C01810=1020.212,130.588,385.207,167.534,51.338,159.515
C01811=1020.208,130.339,385.227,167.532,51.345,159.516
C01812=1020.202,130.090,385.246,167.528,51.352,159.517
C01813=1020.197,129.841,385.267,167.525,51.359,159.518
C01814=1020.191,129.591,385.286,167.522,51.366,159.518
C01815=1020.186,129.343,385.305,167.520,51.373,159.519
C01816=1020.180,129.093,385.324,167.516,51.380,159.520
C01817=1020.175,128.844,385.343,167.513,51.387,159.521
C01818=1020.169,128.595,385.362,167.510,51.394,159.522
C01819=1020.164,128.346,385.381,167.506,51.401,159.522
C01820=1020.158,128.096,385.401,167.504,51.407,159.523
C01821=1020.153,127.847,385.419,167.501,51.415,159.524
C01822=1020.148,127.598,385.439,167.498,51.422,159.525
C01823=1020.142,127.348,385.459,167.495,51.429,159.526
C01824=1020.137,127.099,385.477,167.491,51.436,159.527
C01825=1020.132,126.850,385.497,167.489,51.442,159.528
C01826=1020.126,126.601,385.516,167.486,51.450,159.529
C01827=1020.121,126.352,385.535,167.483,51.457,159.529
C01828=1020.115,126.102,385.554,167.479,51.464,159.530
C01829=1020.109,125.853,385.573,167.477,51.470,159.531
C01830=1020.104,125.604,385.592,167.474,51.477,159.532
C01831=1020.099,125.355,385.611,167.470,51.484,159.533
C01832=1020.094,125.106,385.630,167.467,51.491,159.533
C01833=1020.089,124.856,385.650,167.465,51.498,159.534
C01834=1020.083,124.607,385.669,167.462,51.505,159.535
C01835=1020.078,124.358,385.688,167.459,51.512,159.536
C01836=1020.072,124.109,385.707,167.455,51.519,159.537
C01837=1020.067,123.860,385.726,167.453,51.526,159.538
C01838=1020.061,123.577,385.748,167.449,51.534,159.538
C01839=1020.054,123.294,385.770,167.446,51.541,159.539
C01840=1020.048,123.011,385.792,167.442,51.549,159.540
C01841=1020.042,122.729,385.813,167.439,51.557,159.541
C01842=1020.037,122.480,385.832,167.436,51.564,159.542
C01843=1020.032,122.230,385.852,167.433,51.571,159.543
C01844=1020.027,121.982,385.871,167.430,51.578,159.544
C01845=1020.021,121.732,385.890,167.428,51.585,159.545
C01846=1020.016,121.484,385.909,167.424,51.592,159.545
C01847=1020.010,121.234,385.928,167.421,51.599,159.546
C01848=1020.005,120.985,385.946,167.419,51.606,159.547
C01849=1020.000,120.735,385.965,167.416,51.612,159.548
C01850=1019.994,120.486,385.985,167.412,51.619,159.549
C01851=1019.989,120.237,386.003,167.410,51.626,159.550
C01852=1019.983,119.988,386.023,167.407,51.633,159.550
C01853=1019.978,119.739,386.042,167.403,51.640,159.551
C01854=1019.972,119.490,386.061,167.401,51.647,159.552
C01855=1019.968,119.240,386.080,167.398,51.654,159.553
C01856=1019.963,118.990,386.099,167.395,51.660,159.554
C01857=1019.958,118.742,386.118,167.392,51.667,159.554
C01858=1019.952,118.492,386.137,167.389,51.675,159.555
C01859=1019.947,118.244,386.156,167.386,51.682,159.556
C01860=1019.941,117.993,386.174,167.384,51.688,159.557
C01861=1019.936,117.745,386.193,167.381,51.695,159.558
C01862=1019.931,117.495,386.212,167.377,51.702,159.559
C01863=1019.926,117.247,386.231,167.375,51.709,159.560
C01864=1019.920,116.997,386.251,167.372,51.716,159.560
C01865=1019.915,116.748,386.269,167.369,51.723,159.561
C01866=1019.909,116.498,386.288,167.366,51.729,159.562
C01867=1019.904,116.250,386.307,167.363,51.736,159.563
C01868=1019.899,116.001,386.326,167.361,51.743,159.564
C01869=1019.894,115.751,386.344,167.358,51.750,159.564
C01870=1019.890,115.502,386.364,167.354,51.757,159.565
C01871=1019.884,115.252,386.383,167.352,51.764,159.566
C01872=1019.879,115.004,386.402,167.349,51.771,159.567
C01873=1019.873,114.754,386.420,167.345,51.778,159.568
C01874=1019.868,114.505,386.439,167.343,51.784,159.568
C01875=1019.863,114.255,386.459,167.340,51.791,159.569
C01876=1019.858,114.006,386.477,167.338,51.798,159.570
C01877=1019.853,113.757,386.496,167.334,51.804,159.571
C01878=1019.847,113.508,386.515,167.332,51.811,159.572
C01879=1019.842,113.259,386.533,167.329,51.818,159.572
C01880=1019.837,113.009,386.552,167.325,51.825,159.573
C01881=1019.832,112.760,386.571,167.323,51.831,159.574
C01882=1019.827,112.511,386.589,167.320,51.838,159.575
C01883=1019.821,112.262,386.609,167.318,51.845,159.576
C01884=1019.816,112.012,386.627,167.314,51.852,159.576
C01885=1019.811,111.763,386.646,167.311,51.859,159.577
C01886=1019.806,111.513,386.664,167.309,51.866,159.578
C01887=1019.799,111.264,386.683,167.306,51.873,159.579
C01888=1019.795,111.015,386.701,167.303,51.880,159.580
C01889=1019.790,110.766,386.720,167.301,51.887,159.581
C01890=1019.784,110.516,386.738,167.297,51.894,159.582
C01891=1019.778,110.268,386.757,167.294,51.901,159.582
C01892=1019.774,110.018,386.775,167.292,51.908,159.583
C01893=1019.768,109.769,386.794,167.289,51.915,159.584
C01894=1019.763,109.520,386.812,167.286,51.921,159.585
C01895=1019.757,109.271,386.831,167.283,51.928,159.586
C01896=1019.752,109.021,386.849,167.280,51.935,159.586
C01897=1019.747,108.772,386.867,167.277,51.943,159.587
C01898=1019.741,108.523,386.886,167.275,51.950,159.588
C01899=1019.736,108.273,386.904,167.272,51.957,159.589
C01900=1019.730,108.024,386.922,167.268,51.964,159.590
C01901=1019.725,107.775,386.941,167.266,51.970,159.591
C01902=1019.719,107.492,386.961,167.262,51.978,159.592
C01903=1019.712,107.209,386.982,167.260,51.986,159.593
C01904=1019.706,106.927,387.003,167.257,51.994,159.594
C01905=1019.700,106.644,387.023,167.253,52.002,159.594
C01906=1019.695,106.395,387.041,167.250,52.009,159.595
C01907=1019.689,106.146,387.060,167.248,52.016,159.596
C01908=1019.684,105.896,387.078,167.245,52.023,159.597
C01909=1019.679,105.647,387.096,167.242,52.030,159.598
C01910=1019.674,105.398,387.114,167.239,52.037,159.599
C01911=1019.668,105.148,387.133,167.236,52.044,159.599
C01912=1019.663,104.899,387.151,167.234,52.050,159.600
C01913=1019.658,104.650,387.169,167.231,52.057,159.601
C01914=1019.652,104.400,387.187,167.227,52.064,159.602
C01915=1019.647,104.151,387.206,167.225,52.071,159.603
C01916=1019.641,103.902,387.223,167.222,52.078,159.604
C01917=1019.636,103.652,387.242,167.220,52.085,159.604
C01918=1019.631,103.403,387.260,167.217,52.093,159.605
C01919=1019.625,103.155,387.278,167.214,52.100,159.606
C01920=1019.620,102.905,387.296,167.211,52.106,159.607
C01921=1019.614,102.655,387.314,167.208,52.113,159.608
C01922=1019.609,102.406,387.333,167.206,52.120,159.609
C01923=1019.604,102.157,387.350,167.203,52.127,159.610
C01924=1019.599,101.908,387.369,167.200,52.134,159.610
C01925=1019.593,101.658,387.388,167.197,52.141,159.611
C01926=1019.588,101.409,387.405,167.194,52.148,159.612
C01927=1019.583,101.160,387.423,167.192,52.154,159.613
C01928=1019.578,100.911,387.441,167.189,52.161,159.614
C01929=1019.572,100.661,387.459,167.187,52.168,159.615
C01930=1019.566,100.412,387.478,167.183,52.175,159.615
C01931=1019.562,100.163,387.496,167.180,52.182,159.616
C01932=1019.557,99.914,387.514,167.178,52.189,159.617
C01933=1019.551,99.664,387.532,167.175,52.196,159.618
C01934=1019.546,99.415,387.550,167.173,52.203,159.619
C01935=1019.540,99.166,387.568,167.170,52.210,159.619
C01936=1019.536,98.916,387.586,167.166,52.217,159.620
C01937=1019.529,98.666,387.604,167.164,52.223,159.621
C01938=1019.524,98.417,387.621,167.161,52.230,159.622
C01939=1019.518,98.168,387.639,167.159,52.237,159.623
C01940=1019.514,97.919,387.657,167.156,52.245,159.624
C01941=1019.508,97.670,387.675,167.153,52.252,159.625
C01942=1019.502,97.420,387.693,167.151,52.259,159.625
C01943=1019.496,97.171,387.710,167.147,52.266,159.626
C01944=1019.492,96.922,387.728,167.144,52.273,159.627
C01945=1019.486,96.673,387.746,167.142,52.279,159.628
C01946=1019.481,96.424,387.763,167.139,52.286,159.629
C01947=1019.476,96.173,387.781,167.136,52.293,159.629
C01948=1019.470,95.924,387.799,167.134,52.301,159.630
C01949=1019.465,95.675,387.816,167.131,52.308,159.631
C01950=1019.459,95.426,387.834,167.129,52.315,159.632
C01951=1019.454,95.177,387.852,167.126,52.322,159.633
C01952=1019.448,94.927,387.870,167.122,52.329,159.634
C01953=1019.443,94.678,387.888,167.120,52.335,159.635
C01954=1019.437,94.429,387.905,167.117,52.343,159.635
C01955=1019.432,94.179,387.923,167.115,52.349,159.636
C01956=1019.427,93.930,387.940,167.112,52.356,159.637
C01957=1019.422,93.681,387.958,167.108,52.363,159.638
C01958=1019.417,93.431,387.976,167.106,52.370,159.639
C01959=1019.411,93.182,387.994,167.103,52.377,159.639
C01960=1019.405,92.933,388.011,167.101,52.384,159.640
C01961=1019.400,92.684,388.029,167.098,52.391,159.641
C01962=1019.395,92.434,388.047,167.096,52.398,159.642
C01963=1019.390,92.185,388.064,167.093,52.405,159.643
C01964=1019.384,91.936,388.082,167.090,52.412,159.644
C01965=1019.379,91.687,388.099,167.088,52.419,159.645
C01966=1019.373,91.404,388.119,167.084,52.426,159.645
C01967=1019.367,91.121,388.140,167.081,52.434,159.646
C01968=1019.361,90.839,388.159,167.078,52.442,159.647
C01969=1019.354,90.555,388.179,167.075,52.450,159.648
C01970=1019.349,90.306,388.197,167.072,52.457,159.649
C01971=1019.343,90.057,388.214,167.070,52.464,159.650
C01972=1019.339,89.808,388.233,167.067,52.471,159.651
C01973=1019.333,89.558,388.249,167.064,52.478,159.652
C01974=1019.328,89.309,388.267,167.062,52.485,159.652
C01975=1019.323,89.060,388.285,167.058,52.492,159.653
C01976=1019.317,88.811,388.301,167.056,52.498,159.654
C01977=1019.312,88.561,388.319,167.054,52.506,159.655
C01978=1019.306,88.312,388.337,167.050,52.513,159.656
C01979=1019.301,88.063,388.353,167.048,52.520,159.657
C01980=1019.295,87.813,388.371,167.045,52.527,159.658
C01981=1019.290,87.563,388.388,167.043,52.534,159.658
C01982=1019.284,87.314,388.406,167.040,52.541,159.659
C01983=1019.279,87.065,388.423,167.037,52.548,159.660
C01984=1019.273,86.816,388.440,167.035,52.555,159.661
C01985=1019.268,86.567,388.458,167.032,52.563,159.662
C01986=1019.263,86.317,388.475,167.029,52.570,159.663
C01987=1019.257,86.068,388.492,167.027,52.576,159.664
C01988=1019.252,85.818,388.509,167.023,52.583,159.664
C01989=1019.246,85.569,388.527,167.021,52.590,159.665
C01990=1019.241,85.320,388.543,167.018,52.597,159.666
C01991=1019.236,85.070,388.561,167.015,52.604,159.667
C01992=1019.230,84.821,388.578,167.013,52.611,159.668
C01993=1019.225,84.572,388.595,167.010,52.618,159.668
C01994=1019.220,84.322,388.612,167.008,52.625,159.669
C01995=1019.214,84.073,388.630,167.005,52.633,159.670
C01996=1019.208,83.824,388.646,167.002,52.640,159.671
C01997=1019.203,83.575,388.664,167.000,52.647,159.672
C01998=1019.197,83.325,388.680,166.997,52.654,159.673
C01999=1019.192,83.076,388.698,166.995,52.661,159.674
C02000=1019.187,82.826,388.715,166.991,52.668,159.674
C02001=1019.181,82.577,388.732,166.989,52.674,159.675
C02002=1019.176,82.328,388.749,166.986,52.681,159.676
C02003=1019.171,82.078,388.766,166.983,52.689,159.677
C02004=1019.165,81.829,388.784,166.981,52.695,159.678
C02005=1019.160,81.579,388.801,166.978,52.702,159.679
C02006=1019.155,81.330,388.818,166.976,52.709,159.679
C02007=1019.149,81.081,388.835,166.973,52.716,159.680
C02008=1019.144,80.832,388.853,166.971,52.723,159.681
C02009=1019.139,80.582,388.869,166.967,52.730,159.682
C02010=1019.133,80.332,388.886,166.964,52.737,159.683
C02011=1019.128,80.083,388.904,166.962,52.744,159.684
C02012=1019.123,79.834,388.921,166.959,52.751,159.684
C02013=1019.116,79.585,388.938,166.957,52.758,159.685
C02014=1019.111,79.335,388.955,166.954,52.765,159.686
C02015=1019.106,79.085,388.971,166.952,52.772,159.687
C02016=1019.100,78.836,388.989,166.949,52.779,159.688
C02017=1019.095,78.587,389.006,166.947,52.786,159.689
C02018=1019.091,78.338,389.022,166.943,52.793,159.689
C02019=1019.085,78.089,389.040,166.941,52.800,159.690
C02020=1019.080,77.839,389.057,166.938,52.807,159.691
C02021=1019.075,77.589,389.074,166.936,52.813,159.692
C02022=1019.069,77.340,389.091,166.933,52.821,159.693
C02023=1019.064,77.091,389.108,166.931,52.827,159.694
C02024=1019.058,76.841,389.124,166.928,52.835,159.694
C02025=1019.052,76.592,389.142,166.925,52.842,159.695
C02026=1019.047,76.343,389.159,166.923,52.848,159.696
C02027=1019.042,76.093,389.175,166.920,52.856,159.697
C02028=1019.036,75.844,389.192,166.918,52.862,159.698
C02029=1019.031,75.594,389.209,166.914,52.869,159.699
C02030=1019.025,75.313,389.228,166.912,52.877,159.700
C02031=1019.019,75.030,389.247,166.908,52.886,159.700
C02032=1019.013,74.747,389.266,166.906,52.893,159.701
C02033=1019.007,74.465,389.284,166.903,52.901,159.702
C02034=1019.001,74.215,389.301,166.900,52.908,159.703
C02035=1018.996,73.966,389.318,166.897,52.916,159.704
C02036=1018.991,73.716,389.334,166.895,52.922,159.705
C02037=1018.984,73.467,389.351,166.892,52.929,159.706
C02038=1018.979,73.218,389.368,166.889,52.936,159.706
C02039=1018.974,72.968,389.385,166.886,52.943,159.707
C02040=1018.969,72.719,389.401,166.884,52.950,159.708
C02041=1018.963,72.470,389.418,166.881,52.957,159.709
C02042=1018.957,72.220,389.434,166.878,52.964,159.710
C02043=1018.952,71.971,389.451,166.876,52.971,159.711
C02044=1018.947,71.721,389.468,166.873,52.978,159.711
C02045=1018.941,71.472,389.484,166.871,52.985,159.712
C02046=1018.936,71.223,389.501,166.868,52.992,159.713
C02047=1018.931,70.973,389.517,166.866,52.999,159.714
C02048=1018.925,70.724,389.534,166.863,53.006,159.715
C02049=1018.920,70.474,389.551,166.860,53.013,159.716
C02050=1018.914,70.225,389.567,166.858,53.020,159.716
C02051=1018.909,69.975,389.584,166.855,53.027,159.717
C02052=1018.904,69.726,389.600,166.853,53.034,159.718
C02053=1018.898,69.477,389.616,166.849,53.041,159.719
C02054=1018.893,69.227,389.633,166.847,53.048,159.720
C02055=1018.887,68.978,389.649,166.844,53.055,159.721
C02056=1018.882,68.728,389.666,166.842,53.062,159.721
C02057=1018.877,68.479,389.683,166.839,53.069,159.722
C02058=1018.871,68.230,389.699,166.836,53.076,159.723
C02059=1018.866,67.980,389.716,166.834,53.083,159.724
C02060=1018.860,67.731,389.732,166.831,53.090,159.725
C02061=1018.855,67.481,389.749,166.829,53.097,159.726
C02062=1018.850,67.232,389.765,166.826,53.104,159.726
C02063=1018.844,66.983,389.782,166.823,53.112,159.727
C02064=1018.838,66.733,389.798,166.821,53.118,159.728
C02065=1018.833,66.484,389.814,166.818,53.126,159.729
C02066=1018.828,66.234,389.830,166.816,53.132,159.730
C02067=1018.822,65.985,389.846,166.813,53.140,159.730
C02068=1018.817,65.735,389.863,166.811,53.146,159.731
C02069=1018.811,65.486,389.879,166.808,53.153,159.732
C02070=1018.806,65.237,389.896,166.805,53.161,159.733
C02071=1018.801,64.988,389.912,166.803,53.167,159.734
C02072=1018.795,64.738,389.928,166.800,53.175,159.735
C02073=1018.790,64.488,389.945,166.798,53.181,159.736
C02074=1018.784,64.240,389.960,166.795,53.189,159.736
C02075=1018.779,63.990,389.977,166.791,53.196,159.737
C02076=1018.773,63.741,389.994,166.789,53.203,159.738
C02077=1018.768,63.491,390.009,166.786,53.210,159.739
C02078=1018.763,63.242,390.026,166.784,53.217,159.740
C02079=1018.757,62.992,390.042,166.781,53.224,159.740
C02080=1018.752,62.743,390.059,166.779,53.231,159.741
C02081=1018.746,62.493,390.074,166.776,53.238,159.742
C02082=1018.741,62.244,390.090,166.774,53.246,159.743
C02083=1018.735,61.994,390.106,166.772,53.253,159.744
C02084=1018.729,61.745,390.122,166.769,53.260,159.745
C02085=1018.724,61.496,390.138,166.766,53.267,159.746
C02086=1018.718,61.246,390.153,166.763,53.274,159.746
C02087=1018.712,60.997,390.170,166.761,53.281,159.747
C02088=1018.707,60.747,390.185,166.758,53.288,159.748
C02089=1018.701,60.498,390.201,166.755,53.296,159.749
C02090=1018.696,60.248,390.217,166.753,53.303,159.750
C02091=1018.690,59.998,390.233,166.750,53.310,159.751
C02092=1018.685,59.750,390.249,166.747,53.317,159.752
C02093=1018.679,59.500,390.265,166.745,53.324,159.752
C02094=1018.673,59.232,390.282,166.742,53.332,159.753
C02095=1018.667,58.963,390.299,166.739,53.339,159.754
C02096=1018.661,58.695,390.316,166.737,53.347,159.755
C02097=1018.655,58.426,390.333,166.733,53.355,159.756
C02098=1018.649,58.176,390.349,166.731,53.362,159.757
C02099=1018.644,57.926,390.365,166.728,53.370,159.758
C02100=1018.638,57.678,390.381,166.726,53.376,159.759
C02101=1018.633,57.428,390.396,166.723,53.384,159.759
C02102=1018.627,57.179,390.412,166.720,53.391,159.760
C02103=1018.622,56.929,390.428,166.718,53.398,159.761
C02104=1018.617,56.679,390.444,166.715,53.405,159.762
C02105=1018.612,56.430,390.460,166.712,53.412,159.763
C02106=1018.606,56.180,390.475,166.710,53.419,159.764
C02107=1018.600,55.931,390.491,166.707,53.426,159.764
C02108=1018.595,55.681,390.507,166.704,53.433,159.765
C02109=1018.589,55.432,390.523,166.702,53.440,159.766
C02110=1018.584,55.183,390.538,166.699,53.447,159.767
C02111=1018.578,54.934,390.554,166.697,53.454,159.768
C02112=1018.572,54.684,390.570,166.694,53.461,159.769
C02113=1018.567,54.435,390.586,166.691,53.469,159.769
C02114=1018.561,54.185,390.601,166.689,53.476,159.770
C02115=1018.556,53.936,390.616,166.686,53.483,159.771
C02116=1018.551,53.686,390.633,166.684,53.490,159.772
C02117=1018.545,53.436,390.649,166.681,53.497,159.773
C02118=1018.540,53.187,390.665,166.678,53.504,159.773
C02119=1018.534,52.937,390.680,166.676,53.511,159.774
C02120=1018.529,52.688,390.695,166.673,53.518,159.775
C02121=1018.523,52.439,390.712,166.671,53.525,159.776
C02122=1018.518,52.175,390.728,166.668,53.532,159.777
C02123=1018.511,51.912,390.745,166.665,53.539,159.778
C02124=1018.506,51.649,390.761,166.663,53.547,159.779
C02125=1018.500,51.385,390.778,166.660,53.555,159.779
C02126=1018.495,51.136,390.794,166.657,53.562,159.780
C02127=1018.489,50.886,390.809,166.655,53.569,159.781
C02128=1018.484,50.637,390.824,166.652,53.576,159.782
C02129=1018.478,50.388,390.841,166.650,53.583,159.783
C02130=1018.473,50.138,390.856,166.647,53.590,159.784
C02131=1018.468,49.889,390.871,166.645,53.597,159.784
C02132=1018.462,49.640,390.887,166.642,53.603,159.785
C02133=1018.457,49.390,390.903,166.639,53.611,159.786
C02134=1018.452,49.140,390.918,166.637,53.618,159.787
C02135=1018.447,48.890,390.934,166.634,53.625,159.787
C02136=1018.441,48.642,390.950,166.632,53.632,159.788
C02137=1018.436,48.392,390.965,166.629,53.639,159.789
C02138=1018.431,48.142,390.981,166.627,53.646,159.790
C02139=1018.425,47.893,390.997,166.623,53.652,159.791
C02140=1018.420,47.644,391.012,166.620,53.660,159.791
C02141=1018.414,47.394,391.028,166.618,53.666,159.792
C02142=1018.409,47.145,391.043,166.615,53.674,159.793
C02143=1018.403,46.895,391.059,166.613,53.681,159.794
C02144=1018.398,46.646,391.074,166.611,53.688,159.795
C02145=1018.392,46.396,391.090,166.608,53.694,159.795
C02146=1018.387,46.147,391.105,166.605,53.701,159.796
C02147=1018.381,45.897,391.121,166.603,53.708,159.797
C02148=1018.376,45.648,391.136,166.600,53.715,159.798
C02149=1018.371,45.398,391.152,166.598,53.722,159.799
C02150=1018.366,45.149,391.167,166.595,53.729,159.799
C02151=1018.361,44.900,391.184,166.593,53.736,159.800
C02152=1018.355,44.650,391.199,166.590,53.743,159.801
C02153=1018.350,44.401,391.214,166.588,53.750,159.802
C02154=1018.345,44.151,391.230,166.585,53.756,159.803
C02155=1018.340,43.901,391.245,166.583,53.763,159.803
C02156=1018.335,43.652,391.260,166.580,53.771,159.804
C02157=1018.329,43.403,391.276,166.577,53.778,159.805
C02158=1018.323,43.120,391.294,166.574,53.785,159.806
C02159=1018.317,42.838,391.311,166.571,53.793,159.807
C02160=1018.311,42.554,391.329,166.568,53.800,159.808
C02161=1018.305,42.272,391.347,166.566,53.808,159.809
C02162=1018.300,42.023,391.362,166.563,53.816,159.809
C02163=1018.293,41.773,391.377,166.560,53.823,159.810
C02164=1018.288,41.524,391.392,166.558,53.830,159.811
C02165=1018.283,41.275,391.407,166.555,53.837,159.812
C02166=1018.278,41.025,391.423,166.552,53.844,159.813
C02167=1018.272,40.776,391.437,166.550,53.850,159.813
C02168=1018.266,40.526,391.453,166.547,53.858,159.814
C02169=1018.261,40.276,391.468,166.545,53.865,159.815
C02170=1018.256,40.027,391.482,166.542,53.872,159.816
C02171=1018.250,39.777,391.497,166.539,53.879,159.817
C02172=1018.245,39.528,391.512,166.537,53.886,159.817
C02173=1018.240,39.278,391.528,166.534,53.893,159.818
C02174=1018.234,39.028,391.543,166.532,53.900,159.819
C02175=1018.228,38.779,391.558,166.529,53.907,159.820
C02176=1018.223,38.530,391.573,166.526,53.914,159.820
C02177=1018.218,38.280,391.588,166.524,53.921,159.821
C02178=1018.213,38.031,391.604,166.521,53.928,159.822
C02179=1018.206,37.781,391.619,166.519,53.935,159.823
C02180=1018.201,37.532,391.634,166.516,53.942,159.824
C02181=1018.196,37.283,391.649,166.514,53.949,159.825
C02182=1018.191,37.033,391.664,166.511,53.956,159.825
C02183=1018.185,36.783,391.678,166.508,53.963,159.826
C02184=1018.180,36.534,391.693,166.506,53.970,159.827
C02185=1018.174,36.284,391.709,166.503,53.977,159.828
C02186=1018.169,36.035,391.724,166.501,53.984,159.828
C02187=1018.164,35.785,391.738,166.498,53.991,159.829
C02188=1018.158,35.535,391.753,166.495,53.998,159.830
C02189=1018.152,35.286,391.768,166.493,54.005,159.831
C02190=1018.147,35.037,391.783,166.490,54.013,159.832
C02191=1018.141,34.787,391.798,166.487,54.020,159.832
C02192=1018.136,34.538,391.812,166.486,54.027,159.833
C02193=1018.131,34.288,391.827,166.483,54.034,159.834
C02194=1018.125,34.039,391.842,166.480,54.041,159.835
C02195=1018.119,33.789,391.857,166.478,54.048,159.836
C02196=1018.114,33.540,391.871,166.474,54.055,159.836
C02197=1018.109,33.291,391.886,166.472,54.062,159.837
C02198=1018.103,33.040,391.901,166.470,54.069,159.838
C02199=1018.097,32.791,391.916,166.467,54.076,159.839
C02200=1018.092,32.542,391.930,166.464,54.084,159.840
C02201=1018.087,32.292,391.945,166.462,54.091,159.841
C02202=1018.081,32.043,391.960,166.459,54.098,159.841
C02203=1018.076,31.793,391.975,166.456,54.105,159.842
C02204=1018.070,31.544,391.989,166.454,54.111,159.843
C02205=1018.065,31.295,392.004,166.451,54.119,159.844
C02206=1018.059,31.045,392.019,166.449,54.126,159.845
C02207=1018.054,30.795,392.033,166.446,54.133,159.845
C02208=1018.048,30.546,392.048,166.443,54.140,159.846
C02209=1018.043,30.296,392.063,166.441,54.147,159.847
C02210=1018.038,30.047,392.077,166.438,54.154,159.848
C02211=1018.032,29.797,392.093,166.435,54.161,159.848
C02212=1018.026,29.548,392.107,166.433,54.168,159.849
C02213=1018.021,29.298,392.122,166.430,54.175,159.850
C02214=1018.016,29.049,392.136,166.428,54.182,159.851
C02215=1018.010,28.799,392.151,166.425,54.189,159.852
C02216=1018.005,28.550,392.166,166.422,54.196,159.852
C02217=1018.000,28.300,392.180,166.420,54.203,159.853
C02218=1017.994,28.051,392.195,166.417,54.210,159.854
C02219=1017.989,27.801,392.209,166.415,54.217,159.855
C02220=1017.983,27.551,392.224,166.412,54.224,159.855
C02221=1017.978,27.302,392.239,166.409,54.231,159.856
C02222=1017.972,27.019,392.255,166.407,54.239,159.857
C02223=1017.966,26.736,392.272,166.403,54.247,159.858
C02224=1017.959,26.454,392.288,166.401,54.255,159.859
C02225=1017.953,26.171,392.304,166.398,54.263,159.860
C02226=1017.948,25.922,392.319,166.395,54.270,159.860
C02227=1017.942,25.672,392.333,166.392,54.277,159.861
C02228=1017.937,25.422,392.347,166.390,54.284,159.862
C02229=1017.932,25.173,392.362,166.387,54.292,159.863
C02230=1017.926,24.924,392.376,166.384,54.299,159.864
C02231=1017.920,24.673,392.390,166.383,54.306,159.865
C02232=1017.914,24.424,392.405,166.379,54.312,159.865
C02233=1017.910,24.174,392.419,166.376,54.320,159.866
C02234=1017.904,23.926,392.434,166.375,54.327,159.867
C02235=1017.898,23.676,392.447,166.372,54.334,159.868
C02236=1017.893,23.426,392.461,166.369,54.341,159.868
C02237=1017.888,23.177,392.477,166.366,54.348,159.869
C02238=1017.882,22.928,392.490,166.364,54.355,159.870
C02239=1017.876,22.677,392.505,166.361,54.362,159.871
C02240=1017.870,22.428,392.519,166.359,54.369,159.872
C02241=1017.866,22.178,392.534,166.356,54.377,159.872
C02242=1017.860,21.929,392.548,166.353,54.383,159.873
C02243=1017.855,21.679,392.561,166.351,54.390,159.874
C02244=1017.849,21.430,392.576,166.348,54.398,159.875
C02245=1017.844,21.180,392.590,166.345,54.405,159.875
C02246=1017.839,20.931,392.604,166.343,54.411,159.876
C02247=1017.833,20.682,392.619,166.340,54.419,159.877
C02248=1017.827,20.432,392.633,166.337,54.426,159.878
C02249=1017.823,20.182,392.647,166.335,54.433,159.879
C02250=1017.817,19.932,392.661,166.332,54.440,159.879
C02251=1017.811,19.683,392.676,166.329,54.447,159.880
C02252=1017.805,19.434,392.690,166.327,54.454,159.881
C02253=1017.801,19.184,392.704,166.324,54.461,159.881
C02254=1017.795,18.934,392.718,166.322,54.467,159.882
C02255=1017.790,18.685,392.732,166.319,54.475,159.883
C02256=1017.784,18.436,392.747,166.317,54.482,159.884
C02257=1017.778,18.186,392.760,166.314,54.490,159.885
C02258=1017.773,17.936,392.774,166.311,54.496,159.885
C02259=1017.768,17.687,392.788,166.309,54.503,159.886
C02260=1017.762,17.437,392.802,166.306,54.511,159.887
C02261=1017.757,17.188,392.816,166.304,54.518,159.888
C02262=1017.751,16.938,392.830,166.301,54.524,159.888
C02263=1017.746,16.689,392.845,166.298,54.532,159.889
C02264=1017.741,16.439,392.859,166.296,54.539,159.890
C02265=1017.735,16.190,392.873,166.293,54.546,159.891
C02266=1017.730,15.940,392.887,166.290,54.553,159.891
C02267=1017.724,15.691,392.900,166.288,54.560,159.892
C02268=1017.719,15.441,392.914,166.285,54.567,159.893
C02269=1017.713,15.191,392.928,166.282,54.574,159.894
C02270=1017.708,14.942,392.942,166.280,54.581,159.895
C02271=1017.702,14.692,392.956,166.277,54.588,159.895
C02272=1017.697,14.443,392.970,166.274,54.595,159.896
C02273=1017.691,14.193,392.984,166.272,54.602,159.897
C02274=1017.686,13.944,392.997,166.269,54.609,159.898
C02275=1017.680,13.694,393.011,166.266,54.616,159.898
C02276=1017.676,13.444,393.026,166.264,54.623,159.899
C02277=1017.670,13.195,393.040,166.261,54.630,159.900
C02278=1017.664,12.945,393.053,166.259,54.637,159.901
C02279=1017.658,12.696,393.067,166.256,54.645,159.901
C02280=1017.653,12.446,393.081,166.253,54.651,159.902
C02281=1017.647,12.197,393.095,166.251,54.658,159.903
C02282=1017.642,11.947,393.108,166.248,54.666,159.904
C02283=1017.636,11.698,393.122,166.245,54.673,159.904
C02284=1017.631,11.448,393.135,166.243,54.680,159.905
C02285=1017.625,11.198,393.149,166.240,54.688,159.906
C02286=1017.619,10.918,393.164,166.237,54.695,159.907
C02287=1017.614,10.636,393.179,166.234,54.703,159.908
C02288=1017.607,10.355,393.195,166.231,54.712,159.909
C02289=1017.601,10.074,393.210,166.228,54.719,159.909
C02290=1017.595,9.824,393.224,166.225,54.727,159.910
C02291=1017.590,9.575,393.237,166.222,54.734,159.911
C02292=1017.584,9.325,393.251,166.221,54.741,159.912
C02293=1017.578,9.075,393.264,166.217,54.748,159.912
C02294=1017.573,8.826,393.278,166.215,54.755,159.913
C02295=1017.567,8.576,393.292,166.212,54.763,159.914
C02296=1017.562,8.326,393.305,166.210,54.770,159.915
C02297=1017.556,8.077,393.318,166.207,54.776,159.915
C02298=1017.551,7.828,393.331,166.204,54.784,159.916
C02299=1017.546,7.578,393.345,166.201,54.791,159.917
C02300=1017.540,7.328,393.359,166.199,54.797,159.918
C02301=1017.535,7.079,393.372,166.196,54.805,159.918
C02302=1017.529,6.829,393.386,166.193,54.812,159.919
C02303=1017.523,6.580,393.400,166.192,54.819,159.920
C02304=1017.518,6.330,393.413,166.188,54.826,159.921
C02305=1017.513,6.081,393.426,166.185,54.833,159.922
C02306=1017.508,5.831,393.440,166.183,54.841,159.922
C02307=1017.501,5.582,393.453,166.180,54.847,159.923
C02308=1017.496,5.332,393.466,166.178,54.854,159.924
C02309=1017.491,5.082,393.480,166.175,54.862,159.925
C02310=1017.485,4.833,393.494,166.173,54.868,159.925
C02311=1017.480,4.583,393.506,166.170,54.876,159.926
C02312=1017.475,4.334,393.520,166.167,54.883,159.927
C02313=1017.469,4.084,393.534,166.164,54.890,159.927
C02314=1017.464,3.834,393.547,166.162,54.897,159.928
C02315=1017.458,3.584,393.561,166.159,54.903,159.929
C02316=1017.453,3.336,393.574,166.156,54.911,159.930
C02317=1017.448,3.086,393.587,166.154,54.918,159.931
C02318=1017.442,2.836,393.601,166.151,54.925,159.931
C02319=1017.437,2.586,393.614,166.148,54.932,159.932
C02320=1017.431,2.337,393.627,166.146,54.938,159.933
C02321=1017.426,2.088,393.641,166.143,54.946,159.933
C02322=1017.421,1.838,393.654,166.140,54.953,159.934
C02323=1017.415,1.588,393.668,166.137,54.960,159.935
C02324=1017.409,1.338,393.680,166.135,54.967,159.936
C02325=1017.405,1.089,393.694,166.132,54.974,159.936
C02326=1017.399,0.840,393.708,166.129,54.981,159.937
C02327=1017.394,0.589,393.721,166.127,54.987,159.938
C02328=1017.388,0.340,393.735,166.124,54.995,159.938
C02329=1017.383,0.091,393.747,166.121,55.002,159.939
C02330=1017.378,-0.159,393.761,166.119,55.009,159.940
C02331=1017.372,-0.409,393.774,166.116,55.015,159.940
C02332=1017.367,-0.659,393.788,166.113,55.023,159.941
C02333=1017.362,-0.908,393.800,166.111,55.029,159.942
C02334=1017.356,-1.157,393.814,166.108,55.036,159.943
C02335=1017.351,-1.407,393.828,166.105,55.043,159.943
C02336=1017.346,-1.656,393.841,166.103,55.050,159.944
C02337=1017.340,-1.906,393.854,166.100,55.057,159.945
C02338=1017.335,-2.156,393.867,166.097,55.064,159.945
C02339=1017.330,-2.405,393.881,166.095,55.071,159.946
C02340=1017.325,-2.655,393.894,166.092,55.078,159.947
C02341=1017.318,-2.904,393.907,166.090,55.084,159.948
C02342=1017.313,-3.154,393.920,166.087,55.092,159.948
C02343=1017.309,-3.404,393.933,166.084,55.099,159.949
C02344=1017.303,-3.654,393.947,166.082,55.105,159.950
C02345=1017.298,-3.904,393.960,166.079,55.112,159.950
C02346=1017.292,-4.152,393.973,166.076,55.119,159.951
C02347=1017.287,-4.402,393.986,166.074,55.126,159.952
C02348=1017.281,-4.652,393.999,166.071,55.133,159.952
C02349=1017.277,-4.901,394.012,166.068,55.140,159.953
C02350=1017.270,-5.181,394.026,166.065,55.148,159.954
C02351=1017.264,-5.460,394.041,166.062,55.156,159.955
C02352=1017.258,-5.739,394.055,166.059,55.164,159.956
C02353=1017.252,-6.018,394.070,166.056,55.172,159.956
C02354=1017.246,-6.268,394.082,166.053,55.179,159.957
C02355=1017.241,-6.517,394.095,166.051,55.186,159.958
C02356=1017.236,-6.768,394.108,166.049,55.194,159.959
C02357=1017.230,-7.017,394.120,166.045,55.200,159.959
C02358=1017.224,-7.266,394.133,166.043,55.208,159.960
C02359=1017.219,-7.516,394.146,166.039,55.215,159.960
C02360=1017.214,-7.765,394.159,166.038,55.222,159.961
C02361=1017.208,-8.016,394.172,166.035,55.229,159.962
C02362=1017.203,-8.265,394.184,166.032,55.236,159.963
C02363=1017.197,-8.515,394.196,166.029,55.243,159.964
C02364=1017.192,-8.764,394.210,166.027,55.250,159.964
C02365=1017.186,-9.013,394.223,166.024,55.257,159.965
C02366=1017.181,-9.264,394.236,166.021,55.264,159.966
C02367=1017.176,-9.513,394.248,166.018,55.271,159.966
C02368=1017.170,-9.763,394.260,166.016,55.278,159.967
C02369=1017.165,-10.013,394.274,166.013,55.285,159.968
C02370=1017.160,-10.262,394.286,166.010,55.292,159.968
C02371=1017.154,-10.512,394.300,166.007,55.299,159.969
C02372=1017.149,-10.761,394.312,166.005,55.306,159.970
C02373=1017.143,-11.011,394.324,166.002,55.313,159.971
C02374=1017.138,-11.260,394.337,165.999,55.320,159.971
C02375=1017.132,-11.510,394.350,165.996,55.327,159.972
C02376=1017.127,-11.759,394.362,165.994,55.334,159.973
C02377=1017.122,-12.009,394.375,165.991,55.341,159.973
C02378=1017.116,-12.259,394.388,165.988,55.348,159.974
C02379=1017.111,-12.509,394.400,165.986,55.356,159.975
C02380=1017.106,-12.759,394.413,165.983,55.362,159.975
C02381=1017.100,-13.008,394.425,165.981,55.369,159.976
C02382=1017.095,-13.258,394.438,165.977,55.376,159.977
C02383=1017.090,-13.507,394.450,165.976,55.383,159.978
C02384=1017.084,-13.757,394.463,165.973,55.390,159.978
C02385=1017.079,-14.007,394.476,165.969,55.397,159.979
C02386=1017.073,-14.256,394.489,165.967,55.404,159.979
C02387=1017.069,-14.505,394.502,165.964,55.411,159.980
C02388=1017.063,-14.755,394.514,165.962,55.418,159.981
C02389=1017.057,-15.004,394.527,165.959,55.425,159.981
C02390=1017.053,-15.254,394.539,165.956,55.431,159.982
C02391=1017.047,-15.504,394.552,165.954,55.439,159.983
C02392=1017.042,-15.754,394.563,165.950,55.445,159.983
C02393=1017.037,-16.004,394.577,165.947,55.452,159.984
C02394=1017.031,-16.253,394.589,165.946,55.459,159.985
C02395=1017.025,-16.503,394.601,165.942,55.466,159.985
C02396=1017.020,-16.752,394.613,165.940,55.474,159.986
C02397=1017.014,-17.002,394.626,165.937,55.481,159.987
C02398=1017.009,-17.251,394.638,165.934,55.488,159.988
C02399=1017.004,-17.501,394.650,165.932,55.495,159.988
C02400=1016.999,-17.751,394.663,165.929,55.502,159.989
C02401=1016.993,-18.000,394.675,165.926,55.509,159.990
C02402=1016.988,-18.250,394.688,165.923,55.516,159.990
C02403=1016.982,-18.499,394.700,165.920,55.523,159.991
C02404=1016.977,-18.750,394.712,165.918,55.530,159.992
C02405=1016.971,-18.999,394.724,165.916,55.537,159.993
C02406=1016.966,-19.248,394.736,165.912,55.544,159.993
C02407=1016.960,-19.498,394.749,165.910,55.552,159.994
C02408=1016.955,-19.748,394.760,165.906,55.558,159.994
C02409=1016.949,-19.998,394.773,165.904,55.565,159.995
C02410=1016.944,-20.247,394.785,165.902,55.572,159.996
C02411=1016.940,-20.497,394.797,165.898,55.579,159.996
C02412=1016.934,-20.747,394.809,165.896,55.587,159.997
C02413=1016.928,-20.996,394.822,165.893,55.593,159.998
C02414=1016.922,-21.274,394.835,165.890,55.601,159.998
C02415=1016.916,-21.551,394.848,165.887,55.608,159.999
C02416=1016.910,-21.828,394.861,165.884,55.617,160.000
C02417=1016.905,-22.106,394.876,165.881,55.625,160.001
C02418=1016.900,-22.356,394.887,165.878,55.631,160.001
C02419=1016.894,-22.605,394.900,165.875,55.638,160.002
C02420=1016.888,-22.855,394.912,165.872,55.646,160.003
C02421=1016.883,-23.104,394.924,165.870,55.652,160.003
C02422=1016.878,-23.354,394.936,165.868,55.660,160.004
C02423=1016.872,-23.603,394.948,165.864,55.666,160.005
C02424=1016.867,-23.853,394.960,165.861,55.673,160.005
C02425=1016.862,-24.102,394.972,165.860,55.680,160.006
C02426=1016.856,-24.352,394.985,165.856,55.687,160.007
C02427=1016.851,-24.602,394.996,165.853,55.694,160.007
C02428=1016.846,-24.851,395.008,165.850,55.701,160.008
C02429=1016.841,-25.102,395.021,165.848,55.708,160.009
C02430=1016.835,-25.351,395.033,165.845,55.715,160.009
C02431=1016.830,-25.600,395.045,165.842,55.721,160.010
C02432=1016.825,-25.850,395.056,165.839,55.729,160.011
C02433=1016.819,-26.100,395.069,165.837,55.735,160.011
C02434=1016.814,-26.350,395.080,165.834,55.742,160.012
C02435=1016.809,-26.599,395.093,165.831,55.750,160.013
C02436=1016.804,-26.849,395.104,165.829,55.756,160.013
C02437=1016.798,-27.099,395.117,165.826,55.763,160.014
C02438=1016.793,-27.349,395.128,165.823,55.770,160.014
C02439=1016.788,-27.598,395.140,165.820,55.777,160.015
C02440=1016.782,-27.848,395.152,165.818,55.784,160.016
C02441=1016.777,-28.098,395.164,165.815,55.790,160.016
C02442=1016.772,-28.347,395.176,165.812,55.798,160.017
C02443=1016.767,-28.597,395.187,165.809,55.805,160.018
C02444=1016.761,-28.846,395.199,165.807,55.812,160.018
C02445=1016.755,-29.096,395.211,165.803,55.819,160.019
C02446=1016.750,-29.346,395.223,165.801,55.826,160.020
C02447=1016.745,-29.595,395.234,165.799,55.833,160.020
C02448=1016.740,-29.845,395.246,165.795,55.840,160.021
C02449=1016.733,-30.095,395.258,165.793,55.847,160.022
C02450=1016.728,-30.345,395.269,165.790,55.854,160.022
C02451=1016.723,-30.594,395.281,165.787,55.861,160.023
C02452=1016.718,-30.844,395.293,165.785,55.868,160.024
C02453=1016.713,-31.093,395.304,165.782,55.875,160.024
C02454=1016.707,-31.343,395.315,165.779,55.882,160.025
C02455=1016.701,-31.593,395.327,165.776,55.889,160.026
C02456=1016.696,-31.843,395.339,165.773,55.896,160.026
C02457=1016.691,-32.092,395.351,165.771,55.903,160.027
C02458=1016.686,-32.342,395.362,165.768,55.910,160.028
C02459=1016.680,-32.592,395.373,165.765,55.917,160.028
C02460=1016.675,-32.841,395.385,165.762,55.924,160.029
C02461=1016.670,-33.091,395.397,165.759,55.931,160.029
C02462=1016.665,-33.341,395.409,165.757,55.938,160.030
C02463=1016.659,-33.591,395.420,165.754,55.945,160.031
C02464=1016.653,-33.840,395.432,165.751,55.951,160.031
C02465=1016.648,-34.090,395.443,165.748,55.959,160.032
C02466=1016.643,-34.339,395.455,165.746,55.965,160.033
C02467=1016.638,-34.589,395.466,165.743,55.972,160.033
C02468=1016.632,-34.838,395.478,165.740,55.979,160.034
C02469=1016.627,-35.088,395.489,165.737,55.987,160.034
C02470=1016.622,-35.338,395.501,165.734,55.993,160.035
C02471=1016.617,-35.588,395.513,165.732,56.000,160.036
C02472=1016.611,-35.838,395.523,165.729,56.007,160.036
C02473=1016.606,-36.088,395.535,165.726,56.014,160.037
C02474=1016.601,-36.337,395.547,165.723,56.021,160.037
C02475=1016.596,-36.587,395.559,165.721,56.028,160.038
C02476=1016.591,-36.836,395.570,165.718,56.034,160.039
C02477=1016.585,-37.086,395.581,165.715,56.041,160.039
C02478=1016.579,-37.362,395.594,165.712,56.049,160.040
C02479=1016.573,-37.639,395.606,165.708,56.057,160.041
C02480=1016.568,-37.915,395.619,165.706,56.064,160.041
C02481=1016.562,-38.191,395.632,165.703,56.071,160.042
C02482=1016.557,-38.441,395.643,165.700,56.079,160.043
C02483=1016.552,-38.690,395.655,165.697,56.086,160.043
C02484=1016.547,-38.940,395.666,165.695,56.092,160.044
C02485=1016.541,-39.190,395.677,165.692,56.099,160.044
C02486=1016.536,-39.440,395.688,165.689,56.106,160.045
C02487=1016.531,-39.689,395.700,165.685,56.113,160.045
C02488=1016.525,-39.939,395.711,165.683,56.120,160.046
C02489=1016.520,-40.189,395.722,165.681,56.127,160.047
C02490=1016.515,-40.438,395.733,165.678,56.134,160.047
C02491=1016.510,-40.688,395.745,165.675,56.140,160.048
C02492=1016.504,-40.937,395.755,165.672,56.148,160.049
C02493=1016.499,-41.187,395.767,165.669,56.155,160.049
C02494=1016.493,-41.437,395.778,165.666,56.162,160.050
C02495=1016.488,-41.687,395.789,165.663,56.169,160.050
C02496=1016.483,-41.937,395.799,165.661,56.176,160.051
C02497=1016.478,-42.186,395.811,165.658,56.183,160.052
C02498=1016.472,-42.436,395.822,165.655,56.189,160.052
C02499=1016.467,-42.686,395.833,165.652,56.196,160.053
C02500=1016.461,-42.935,395.844,165.649,56.204,160.054
C02501=1016.456,-43.185,395.856,165.647,56.210,160.054
C02502=1016.451,-43.435,395.866,165.644,56.217,160.055
C02503=1016.446,-43.685,395.877,165.641,56.224,160.055
C02504=1016.440,-43.934,395.888,165.638,56.231,160.056
C02505=1016.435,-44.184,395.900,165.635,56.238,160.057
C02506=1016.429,-44.434,395.910,165.633,56.245,160.057
C02507=1016.425,-44.684,395.921,165.630,56.252,160.058
C02508=1016.420,-44.933,395.932,165.627,56.259,160.058
C02509=1016.415,-45.183,395.943,165.624,56.266,160.059
C02510=1016.409,-45.432,395.954,165.621,56.272,160.059
C02511=1016.404,-45.682,395.966,165.619,56.279,160.060
C02512=1016.398,-45.932,395.976,165.615,56.286,160.061
C02513=1016.393,-46.182,395.987,165.613,56.293,160.061
C02514=1016.388,-46.431,395.998,165.610,56.300,160.062
C02515=1016.383,-46.681,396.010,165.608,56.307,160.063
C02516=1016.377,-46.931,396.020,165.605,56.314,160.063
C02517=1016.373,-47.180,396.031,165.602,56.320,160.064
C02518=1016.367,-47.430,396.042,165.598,56.327,160.064
C02519=1016.361,-47.679,396.053,165.595,56.334,160.065
C02520=1016.357,-47.930,396.063,165.593,56.341,160.065
C02521=1016.351,-48.179,396.074,165.590,56.348,160.066
C02522=1016.346,-48.429,396.086,165.587,56.354,160.066
C02523=1016.341,-48.679,396.095,165.584,56.361,160.067
C02524=1016.336,-48.928,396.107,165.582,56.368,160.068
C02525=1016.330,-49.178,396.118,165.579,56.375,160.068
C02526=1016.326,-49.428,396.129,165.576,56.382,160.069
C02527=1016.320,-49.678,396.139,165.574,56.388,160.069
C02528=1016.315,-49.927,396.151,165.571,56.395,160.070
C02529=1016.310,-50.177,396.161,165.568,56.402,160.070
C02530=1016.305,-50.427,396.172,165.564,56.409,160.071
C02531=1016.300,-50.677,396.182,165.562,56.415,160.072
C02532=1016.295,-50.927,396.194,165.559,56.422,160.072
C02533=1016.289,-51.176,396.205,165.556,56.429,160.073
C02534=1016.283,-51.426,396.215,165.553,56.436,160.073
C02535=1016.279,-51.676,396.225,165.551,56.443,160.074
C02536=1016.273,-51.925,396.236,165.548,56.450,160.074
C02537=1016.267,-52.175,396.246,165.545,56.457,160.075
C02538=1016.262,-52.425,396.257,165.543,56.464,160.076
C02539=1016.258,-52.674,396.267,165.540,56.471,160.076
C02540=1016.252,-52.925,396.277,165.537,56.478,160.077
C02541=1016.246,-53.174,396.288,165.534,56.485,160.077
C02542=1016.241,-53.451,396.299,165.530,56.493,160.078
C02543=1016.235,-53.728,396.310,165.528,56.501,160.079
C02544=1016.228,-54.004,396.322,165.524,56.509,160.079
C02545=1016.223,-54.281,396.333,165.521,56.516,160.080
C02546=1016.217,-54.530,396.344,165.518,56.523,160.081
C02547=1016.212,-54.780,396.354,165.515,56.530,160.081
C02548=1016.207,-55.030,396.364,165.512,56.537,160.082
C02549=1016.201,-55.279,396.375,165.509,56.544,160.082
C02550=1016.196,-55.529,396.385,165.507,56.551,160.083
C02551=1016.191,-55.779,396.395,165.505,56.558,160.084
C02552=1016.186,-56.029,396.405,165.501,56.565,160.084
C02553=1016.181,-56.279,396.416,165.498,56.572,160.085
C02554=1016.175,-56.529,396.426,165.495,56.579,160.085
C02555=1016.170,-56.778,396.436,165.492,56.586,160.086
C02556=1016.165,-57.028,396.446,165.489,56.593,160.086
C02557=1016.159,-57.278,396.457,165.487,56.599,160.087
C02558=1016.154,-57.527,396.467,165.484,56.606,160.088
C02559=1016.149,-57.777,396.477,165.481,56.613,160.088
C02560=1016.144,-58.027,396.487,165.479,56.621,160.089
C02561=1016.138,-58.276,396.498,165.475,56.628,160.089
C02562=1016.133,-58.526,396.508,165.472,56.634,160.090
C02563=1016.128,-58.776,396.518,165.470,56.641,160.091
C02564=1016.123,-59.026,396.528,165.467,56.648,160.091
C02565=1016.117,-59.276,396.538,165.464,56.655,160.092
C02566=1016.112,-59.525,396.549,165.461,56.662,160.092
C02567=1016.107,-59.775,396.559,165.458,56.669,160.093
C02568=1016.101,-60.025,396.569,165.456,56.675,160.093
C02569=1016.097,-60.274,396.579,165.453,56.682,160.094
C02570=1016.092,-60.525,396.590,165.450,56.689,160.094
C02571=1016.087,-60.774,396.599,165.447,56.696,160.095
C02572=1016.081,-61.024,396.610,165.444,56.703,160.095
C02573=1016.076,-61.273,396.620,165.442,56.709,160.096
C02574=1016.071,-61.523,396.630,165.439,56.716,160.097
C02575=1016.066,-61.773,396.640,165.436,56.723,160.097
C02576=1016.061,-62.023,396.650,165.432,56.729,160.097
C02577=1016.055,-62.273,396.660,165.430,56.736,160.098
C02578=1016.050,-62.522,396.670,165.427,56.743,160.099
C02579=1016.045,-62.772,396.680,165.424,56.750,160.099
C02580=1016.040,-63.022,396.690,165.421,56.757,160.100
C02581=1016.034,-63.271,396.701,165.419,56.763,160.100
C02582=1016.030,-63.521,396.711,165.416,56.770,160.101
C02583=1016.024,-63.771,396.721,165.413,56.777,160.101
C02584=1016.019,-64.020,396.731,165.410,56.784,160.102
C02585=1016.014,-64.270,396.741,165.408,56.790,160.102
C02586=1016.009,-64.520,396.751,165.404,56.797,160.103
C02587=1016.004,-64.770,396.761,165.401,56.804,160.103
C02588=1015.999,-65.019,396.771,165.398,56.811,160.104
C02589=1015.993,-65.269,396.781,165.396,56.817,160.104
C02590=1015.989,-65.519,396.791,165.393,56.824,160.105
C02591=1015.983,-65.769,396.801,165.390,56.831,160.105
C02592=1015.978,-66.018,396.811,165.387,56.837,160.106
C02593=1015.973,-66.268,396.821,165.385,56.844,160.106
C02594=1015.968,-66.518,396.831,165.382,56.851,160.107
C02595=1015.963,-66.768,396.841,165.379,56.858,160.107
C02596=1015.958,-67.017,396.851,165.377,56.864,160.108
C02597=1015.954,-67.267,396.861,165.373,56.870,160.108
C02598=1015.948,-67.517,396.871,165.370,56.877,160.109
C02599=1015.943,-67.766,396.881,165.368,56.884,160.110
C02600=1015.938,-68.016,396.891,165.365,56.891,160.110
C02601=1015.933,-68.266,396.901,165.361,56.897,160.110
C02602=1015.928,-68.516,396.911,165.359,56.903,160.111
C02603=1015.923,-68.765,396.921,165.356,56.910,160.111
C02604=1015.918,-69.015,396.930,165.353,56.917,160.112
C02605=1015.913,-69.266,396.940,165.351,56.923,160.112
C02606=1015.907,-69.543,396.951,165.347,56.930,160.113
C02607=1015.902,-69.821,396.962,165.344,56.938,160.114
C02608=1015.896,-70.098,396.973,165.341,56.945,160.114
C02609=1015.890,-70.376,396.983,165.337,56.952,160.114
C02610=1015.885,-70.626,396.994,165.335,56.959,160.115
C02611=1015.880,-70.876,397.003,165.332,56.966,160.116
C02612=1015.875,-71.125,397.013,165.330,56.972,160.116
C02613=1015.870,-71.375,397.023,165.327,56.979,160.116
C02614=1015.865,-71.625,397.033,165.324,56.986,160.117
C02615=1015.861,-71.875,397.042,165.321,56.991,160.117
C02616=1015.855,-72.125,397.052,165.318,56.998,160.118
C02617=1015.850,-72.374,397.062,165.314,57.005,160.118
C02618=1015.845,-72.624,397.072,165.312,57.011,160.119
C02619=1015.840,-72.874,397.082,165.309,57.018,160.119
C02620=1015.836,-73.124,397.091,165.307,57.024,160.120
C02621=1015.831,-73.373,397.101,165.304,57.031,160.120
C02622=1015.825,-73.623,397.111,165.300,57.037,160.120
C02623=1015.820,-73.873,397.121,165.298,57.044,160.121
C02624=1015.816,-74.122,397.131,165.295,57.050,160.121
C02625=1015.811,-74.372,397.140,165.293,57.056,160.122
C02626=1015.806,-74.622,397.150,165.289,57.063,160.122
C02627=1015.801,-74.872,397.160,165.286,57.070,160.123
C02628=1015.796,-75.122,397.169,165.284,57.076,160.124
C02629=1015.791,-75.372,397.179,165.281,57.083,160.124
C02630=1015.786,-75.622,397.188,165.278,57.089,160.124
C02631=1015.781,-75.871,397.197,165.275,57.096,160.125
C02632=1015.776,-76.120,397.207,165.273,57.103,160.125
C02633=1015.770,-76.371,397.216,165.270,57.110,160.126
C02634=1015.765,-76.620,397.226,165.266,57.116,160.126
C02635=1015.761,-76.870,397.235,165.264,57.123,160.127
C02636=1015.756,-77.120,397.245,165.261,57.130,160.127
C02637=1015.750,-77.370,397.254,165.258,57.136,160.128
C02638=1015.745,-77.620,397.263,165.256,57.142,160.128
C02639=1015.741,-77.870,397.272,165.253,57.149,160.129
C02640=1015.735,-78.119,397.282,165.249,57.156,160.129
C02641=1015.731,-78.369,397.291,165.247,57.162,160.130
C02642=1015.725,-78.619,397.301,165.244,57.169,160.130
C02643=1015.720,-78.868,397.309,165.241,57.175,160.130
C02644=1015.715,-79.118,397.319,165.239,57.182,160.131
C02645=1015.710,-79.368,397.328,165.236,57.189,160.132
C02646=1015.706,-79.617,397.338,165.232,57.195,160.132
C02647=1015.700,-79.867,397.346,165.230,57.202,160.133
C02648=1015.695,-80.118,397.356,165.227,57.208,160.133
C02649=1015.690,-80.367,397.366,165.224,57.215,160.133
C02650=1015.685,-80.617,397.374,165.222,57.221,160.134
C02651=1015.680,-80.866,397.384,165.218,57.228,160.134
C02652=1015.675,-81.116,397.392,165.215,57.235,160.135
C02653=1015.670,-81.366,397.401,165.212,57.242,160.135
C02654=1015.665,-81.616,397.410,165.210,57.248,160.136
C02655=1015.659,-81.866,397.420,165.207,57.255,160.136
C02656=1015.655,-82.116,397.429,165.204,57.261,160.137
C02657=1015.649,-82.365,397.437,165.201,57.268,160.137
C02658=1015.645,-82.615,397.446,165.199,57.275,160.138
C02659=1015.639,-82.864,397.455,165.195,57.281,160.138
C02660=1015.634,-83.114,397.464,165.192,57.288,160.139
C02661=1015.629,-83.364,397.473,165.189,57.295,160.139
///RCONF 1,0,0,0,1,0,0,0,0,0,0,0,0,0,0,0,0,0,0,0,0,0,0,0
C02662=1015.624,-83.614,397.481,165.187,57.302,160.140
C02663=1015.620,-83.864,397.491,165.184,57.308,160.140
C02664=1015.613,-84.114,397.500,165.181,57.315,160.141
C02665=1015.608,-84.363,397.509,165.179,57.322,160.141
C02666=1015.604,-84.613,397.518,165.175,57.328,160.141
C02667=1015.598,-84.863,397.526,165.172,57.335,160.142
C02668=1015.594,-85.113,397.535,165.170,57.341,160.143
C02669=1015.589,-85.363,397.544,165.167,57.348,160.143
C02670=1015.584,-85.584,397.551,165.164,57.354,160.143
C02671=1015.580,-85.806,397.560,165.162,57.359,160.144
C02672=1015.575,-86.028,397.567,165.159,57.365,160.144
C02673=1015.570,-86.249,397.575,165.157,57.371,160.145
C02674=1015.567,-86.471,397.583,165.154,57.377,160.145
C02675=1015.562,-86.692,397.591,165.152,57.383,160.145
C02676=1015.558,-86.913,397.598,165.149,57.389,160.146
C02677=1015.553,-87.135,397.607,165.147,57.394,160.146
C02678=1015.548,-87.385,397.615,165.143,57.401,160.146
C02679=1015.543,-87.635,397.625,165.140,57.408,160.147
C02680=1015.538,-87.885,397.633,165.139,57.414,160.148
C02681=1015.532,-88.134,397.642,165.135,57.421,160.148
C02682=1015.528,-88.384,397.651,165.132,57.428,160.148
C02683=1015.523,-88.633,397.659,165.130,57.433,160.149
C02684=1015.519,-88.883,397.669,165.127,57.440,160.149
C02685=1015.513,-89.133,397.677,165.124,57.446,160.150
C02686=1015.508,-89.382,397.685,165.121,57.453,160.150
C02687=1015.504,-89.632,397.695,165.118,57.460,160.150
C02688=1015.498,-89.882,397.703,165.116,57.466,160.151
C02689=1015.494,-90.132,397.712,165.112,57.472,160.151
C02690=1015.489,-90.382,397.721,165.109,57.479,160.152
C02691=1015.483,-90.632,397.729,165.107,57.485,160.152
C02692=1015.479,-90.882,397.738,165.103,57.492,160.152
C02693=1015.474,-91.131,397.747,165.101,57.498,160.153
C02694=1015.469,-91.381,397.756,165.098,57.504,160.153
C02695=1015.464,-91.631,397.764,165.096,57.511,160.154
C02696=1015.459,-91.881,397.773,165.092,57.517,160.154
C02697=1015.454,-92.131,397.782,165.089,57.524,160.155
C02698=1015.449,-92.381,397.790,165.087,57.530,160.155
C02699=1015.445,-92.630,397.799,165.083,57.536,160.155
C02700=1015.440,-92.880,397.807,165.082,57.543,160.156
C02701=1015.434,-93.129,397.816,165.078,57.549,160.156
C02702=1015.430,-93.380,397.824,165.076,57.555,160.157
C02703=1015.425,-93.630,397.833,165.073,57.562,160.157
C02704=1015.420,-93.879,397.841,165.070,57.568,160.158
C02705=1015.415,-94.129,397.850,165.067,57.574,160.158
C02706=1015.410,-94.378,397.859,165.065,57.581,160.159
C02707=1015.406,-94.628,397.868,165.061,57.587,160.159
C02708=1015.401,-94.878,397.876,165.059,57.593,160.159
C02709=1015.395,-95.128,397.885,165.056,57.600,160.160
C02710=1015.390,-95.464,397.896,165.052,57.608,160.160
C02711=1015.383,-95.801,397.908,165.048,57.617,160.161
C02712=1015.376,-96.137,397.919,165.044,57.625,160.161
C02713=1015.369,-96.473,397.931,165.041,57.633,160.162
C02714=1015.365,-96.724,397.939,165.037,57.640,160.162
C02715=1015.360,-96.973,397.947,165.035,57.645,160.162
C02716=1015.355,-97.222,397.956,165.032,57.652,160.163
C02717=1015.351,-97.472,397.965,165.030,57.658,160.163
C02718=1015.345,-97.722,397.973,165.026,57.665,160.164
C02719=1015.341,-97.973,397.982,165.024,57.671,160.164
C02720=1015.336,-98.222,397.990,165.021,57.678,160.164
C02721=1015.331,-98.472,397.998,165.018,57.683,160.165
C02722=1015.326,-98.722,398.006,165.015,57.690,160.165
C02723=1015.321,-98.972,398.015,165.013,57.696,160.166
C02724=1015.316,-99.221,398.023,165.009,57.703,160.166
C02725=1015.311,-99.471,398.030,165.006,57.710,160.166
C02726=1015.306,-99.721,398.039,165.004,57.716,160.167
C02727=1015.301,-99.971,398.047,165.000,57.722,160.167
C02728=1015.297,-100.220,398.055,164.998,57.728,160.168
C02729=1015.292,-100.471,398.063,164.995,57.735,160.168
C02730=1015.287,-100.720,398.072,164.993,57.741,160.168
C02731=1015.282,-100.970,398.080,164.990,57.748,160.169
C02732=1015.277,-101.220,398.088,164.987,57.754,160.169
C02733=1015.272,-101.469,398.096,164.984,57.760,160.170
C02734=1015.267,-101.751,398.105,164.981,57.767,160.170
C02735=1015.262,-102.033,398.114,164.978,57.774,160.170
C02736=1015.256,-102.315,398.123,164.975,57.781,160.171
C02737=1015.250,-102.597,398.132,164.971,57.788,160.171
C02738=1015.246,-102.846,398.141,164.968,57.794,160.172
C02739=1015.241,-103.097,398.148,164.965,57.801,160.172
C02740=1015.236,-103.346,398.157,164.963,57.807,160.173
C02741=1015.231,-103.596,398.164,164.960,57.814,160.173
C02742=1015.226,-103.846,398.173,164.957,57.819,160.173
C02743=1015.221,-104.096,398.181,164.955,57.825,160.174
C02744=1015.217,-104.345,398.189,164.952,57.832,160.174
C02745=1015.212,-104.595,398.196,164.949,57.838,160.175
C02746=1015.207,-104.844,398.205,164.946,57.845,160.175
C02747=1015.202,-105.095,398.212,164.943,57.850,160.175
C02748=1015.197,-105.345,398.220,164.940,57.857,160.175
C02749=1015.192,-105.594,398.228,164.938,57.863,160.176
C02750=1015.187,-105.844,398.236,164.934,57.870,160.176
C02751=1015.183,-106.094,398.245,164.932,57.876,160.177
C02752=1015.178,-106.344,398.253,164.930,57.882,160.177
C02753=1015.174,-106.594,398.260,164.926,57.888,160.177
C02754=1015.169,-106.843,398.268,164.924,57.894,160.178
C02755=1015.164,-107.094,398.276,164.921,57.901,160.178
C02756=1015.159,-107.343,398.284,164.918,57.907,160.179
C02757=1015.154,-107.593,398.292,164.915,57.913,160.179
C02758=1015.149,-107.843,398.300,164.912,57.919,160.179
C02759=1015.145,-108.093,398.307,164.910,57.925,160.180
C02760=1015.140,-108.343,398.316,164.906,57.931,160.180
C02761=1015.135,-108.592,398.323,164.904,57.937,160.180
C02762=1015.130,-108.842,398.330,164.901,57.944,160.181
C02763=1015.125,-109.092,398.338,164.899,57.950,160.181
C02764=1015.120,-109.342,398.346,164.895,57.956,160.181
C02765=1015.116,-109.591,398.354,164.893,57.962,160.182
C02766=1015.111,-109.842,398.361,164.889,57.969,160.182
C02767=1015.106,-110.091,398.369,164.887,57.975,160.183
C02768=1015.101,-110.342,398.377,164.885,57.981,160.183
C02769=1015.096,-110.590,398.384,164.882,57.987,160.183
C02770=1015.091,-110.841,398.392,164.879,57.993,160.184
C02771=1015.087,-111.090,398.399,164.876,58.000,160.184
C02772=1015.082,-111.341,398.407,164.873,58.006,160.184
C02773=1015.077,-111.590,398.414,164.871,58.011,160.185
C02774=1015.072,-111.841,398.422,164.867,58.018,160.185
C02775=1015.068,-112.090,398.430,164.865,58.024,160.185
C02776=1015.063,-112.340,398.438,164.861,58.030,160.185
C02777=1015.058,-112.589,398.445,164.860,58.037,160.186
C02778=1015.053,-112.840,398.453,164.857,58.043,160.187
C02779=1015.048,-113.089,398.460,164.854,58.049,160.187
C02780=1015.044,-113.339,398.467,164.851,58.055,160.187
C02781=1015.039,-113.589,398.475,164.849,58.061,160.188
C02782=1015.035,-113.839,398.483,164.845,58.067,160.188
C02783=1015.030,-114.089,398.490,164.843,58.073,160.188
C02784=1015.025,-114.338,398.498,164.840,58.079,160.189
C02785=1015.020,-114.588,398.505,164.837,58.085,160.189
C02786=1015.015,-114.838,398.513,164.835,58.091,160.189
C02787=1015.011,-115.088,398.520,164.832,58.097,160.190
C02788=1015.006,-115.338,398.528,164.829,58.103,160.190
C02789=1015.001,-115.588,398.536,164.826,58.109,160.190
C02790=1014.996,-115.837,398.542,164.824,58.115,160.191
C02791=1014.992,-116.088,398.550,164.820,58.121,160.191
C02792=1014.987,-116.337,398.557,164.818,58.127,160.191
C02793=1014.982,-116.588,398.565,164.816,58.133,160.192
C02794=1014.977,-116.837,398.571,164.812,58.140,160.192
C02795=1014.973,-117.087,398.579,164.810,58.146,160.192
C02796=1014.968,-117.337,398.587,164.807,58.151,160.193
C02797=1014.964,-117.587,398.594,164.804,58.158,160.193
C02798=1014.958,-117.869,398.603,164.800,58.164,160.193
C02799=1014.953,-118.151,398.610,164.797,58.171,160.193
C02800=1014.947,-118.432,398.618,164.795,58.178,160.194
C02801=1014.941,-118.714,398.627,164.791,58.185,160.194
C02802=1014.937,-118.964,398.634,164.789,58.191,160.195
C02803=1014.933,-119.214,398.641,164.786,58.197,160.195
C02804=1014.928,-119.463,398.648,164.783,58.203,160.195
C02805=1014.923,-119.714,398.656,164.780,58.209,160.196
C02806=1014.918,-119.963,398.663,164.778,58.215,160.196
C02807=1014.914,-120.213,398.670,164.776,58.221,160.196
C02808=1014.909,-120.464,398.677,164.772,58.227,160.197
C02809=1014.904,-120.713,398.684,164.770,58.233,160.197
C02810=1014.900,-120.963,398.692,164.767,58.238,160.197
C02811=1014.895,-121.212,398.699,164.764,58.244,160.197
C02812=1014.890,-121.463,398.706,164.761,58.250,160.198
C02813=1014.886,-121.713,398.713,164.758,58.256,160.198
C02814=1014.881,-121.962,398.720,164.756,58.262,160.198
C02815=1014.876,-122.212,398.727,164.754,58.268,160.199
C02816=1014.871,-122.462,398.735,164.750,58.274,160.199
C02817=1014.866,-122.712,398.741,164.748,58.280,160.199
C02818=1014.862,-122.962,398.748,164.745,58.286,160.200
C02819=1014.858,-123.211,398.756,164.742,58.292,160.200
C02820=1014.852,-123.462,398.762,164.740,58.297,160.200
C02821=1014.848,-123.712,398.770,164.737,58.304,160.201
C02822=1014.843,-123.961,398.777,164.734,58.310,160.201
C02823=1014.839,-124.211,398.784,164.731,58.315,160.201
C02824=1014.835,-124.461,398.791,164.729,58.321,160.201
C02825=1014.829,-124.711,398.798,164.726,58.327,160.202
C02826=1014.825,-124.961,398.805,164.723,58.333,160.202
C02827=1014.820,-125.210,398.811,164.720,58.339,160.202
C02828=1014.815,-125.460,398.819,164.717,58.344,160.203
C02829=1014.811,-125.710,398.825,164.715,58.350,160.203
C02830=1014.806,-125.960,398.832,164.713,58.356,160.203
C02831=1014.801,-126.210,398.839,164.709,58.362,160.204
C02832=1014.796,-126.460,398.846,164.707,58.368,160.204
C02833=1014.792,-126.710,398.852,164.704,58.374,160.204
C02834=1014.787,-126.959,398.860,164.701,58.380,160.204
C02835=1014.782,-127.209,398.866,164.699,58.385,160.205
C02836=1014.778,-127.459,398.873,164.696,58.392,160.205
C02837=1014.774,-127.709,398.880,164.693,58.398,160.205
C02838=1014.769,-127.959,398.887,164.690,58.403,160.206
C02839=1014.764,-128.208,398.893,164.688,58.409,160.206
C02840=1014.760,-128.458,398.901,164.685,58.414,160.206
C02841=1014.756,-128.708,398.909,164.683,58.419,160.206
C02842=1014.752,-128.957,398.917,164.679,58.423,160.206
C02843=1014.749,-129.206,398.927,164.678,58.427,160.206
C02844=1014.746,-129.456,398.936,164.675,58.430,160.206
C02845=1014.744,-129.706,398.947,164.673,58.433,160.206
C02846=1014.741,-129.956,398.957,164.670,58.435,160.206
C02847=1014.740,-130.205,398.970,164.668,58.436,160.205
C02848=1014.738,-130.455,398.982,164.666,58.437,160.205
C02849=1014.737,-130.704,398.994,164.664,58.438,160.204
C02850=1014.736,-130.954,399.007,164.661,58.438,160.203
C02851=1014.736,-131.204,399.021,164.659,58.437,160.203
C02852=1014.736,-131.454,399.036,164.656,58.436,160.202
C02853=1014.736,-131.703,399.051,164.655,58.434,160.201
C02854=1014.737,-131.953,399.067,164.653,58.431,160.200
C02855=1014.738,-132.202,399.083,164.651,58.429,160.199
C02856=1014.740,-132.452,399.100,164.649,58.425,160.198
C02857=1014.741,-132.702,399.117,164.646,58.422,160.196
C02858=1014.744,-132.951,399.136,164.645,58.416,160.195
C02859=1014.747,-133.201,399.154,164.643,58.412,160.194
C02860=1014.749,-133.451,399.173,164.641,58.406,160.192
C02861=1014.752,-133.700,399.193,164.639,58.400,160.190
C02862=1014.514,-133.726,398.785,164.611,58.759,160.248
C02863=1014.510,-133.477,398.765,164.613,58.764,160.249
C02864=1014.508,-133.227,398.746,164.615,58.770,160.251
C02865=1014.505,-132.978,398.727,164.617,58.775,160.252
C02866=1014.503,-132.728,398.709,164.619,58.780,160.254
C02867=1014.501,-132.478,398.692,164.620,58.783,160.255
C02868=1014.500,-132.229,398.674,164.623,58.786,160.256
C02869=1014.499,-131.979,398.658,164.625,58.789,160.257
C02870=1014.498,-131.729,398.642,164.627,58.792,160.258
C02871=1014.498,-131.480,398.627,164.629,58.794,160.259
C02872=1014.498,-131.229,398.612,164.631,58.795,160.260
C02873=1014.499,-130.980,398.599,164.633,58.795,160.261
C02874=1014.499,-130.730,398.585,164.635,58.796,160.261
C02875=1014.500,-130.481,398.572,164.637,58.796,160.262
C02876=1014.502,-130.231,398.560,164.640,58.795,160.262
C02877=1014.503,-129.981,398.549,164.642,58.793,160.263
C02878=1014.506,-129.732,398.538,164.645,58.790,160.263
C02879=1014.507,-129.482,398.528,164.648,58.788,160.264
C02880=1014.511,-129.233,398.518,164.650,58.786,160.264
C02881=1014.514,-128.984,398.509,164.652,58.782,160.264
C02882=1014.517,-128.734,398.501,164.655,58.778,160.264
C02883=1014.521,-128.484,398.493,164.656,58.773,160.263
C02884=1014.525,-128.234,398.485,164.659,58.768,160.263
C02885=1014.530,-127.985,398.478,164.662,58.762,160.263
C02886=1014.535,-127.735,398.471,164.665,58.756,160.263
C02887=1014.539,-127.485,398.465,164.667,58.750,160.262
C02888=1014.544,-127.236,398.457,164.671,58.745,160.262
C02889=1014.549,-126.986,398.451,164.673,58.739,160.262
C02890=1014.553,-126.736,398.444,164.676,58.733,160.262
C02891=1014.558,-126.486,398.438,164.679,58.728,160.261
C02892=1014.562,-126.237,398.430,164.681,58.722,160.261
C02893=1014.567,-125.987,398.424,164.683,58.716,160.261
C02894=1014.572,-125.736,398.417,164.686,58.710,160.260
C02895=1014.577,-125.486,398.411,164.690,58.704,160.260
C02896=1014.581,-125.237,398.403,164.692,58.698,160.260
C02897=1014.586,-124.987,398.397,164.694,58.692,160.259
C02898=1014.590,-124.737,398.390,164.697,58.686,160.259
C02899=1014.595,-124.488,398.383,164.700,58.681,160.259
C02900=1014.599,-124.238,398.376,164.702,58.675,160.259
C02901=1014.604,-123.987,398.368,164.704,58.669,160.258
C02902=1014.609,-123.738,398.362,164.708,58.663,160.258
C02903=1014.613,-123.488,398.355,164.711,58.657,160.258
C02904=1014.618,-123.238,398.347,164.713,58.651,160.257
C02905=1014.623,-122.989,398.341,164.716,58.646,160.257
C02906=1014.627,-122.738,398.334,164.718,58.640,160.257
C02907=1014.632,-122.488,398.326,164.721,58.634,160.256
C02908=1014.637,-122.239,398.319,164.724,58.628,160.256
C02909=1014.641,-121.988,398.313,164.727,58.623,160.256
C02910=1014.645,-121.739,398.305,164.729,58.617,160.256
C02911=1014.650,-121.490,398.298,164.732,58.611,160.255
C02912=1014.655,-121.239,398.291,164.734,58.605,160.255
C02913=1014.659,-120.989,398.284,164.738,58.598,160.255
C02914=1014.665,-120.740,398.277,164.740,58.593,160.255
C02915=1014.669,-120.490,398.270,164.743,58.587,160.254
C02916=1014.674,-120.240,398.262,164.745,58.581,160.254
C02917=1014.679,-119.990,398.256,164.748,58.575,160.253
C02918=1014.683,-119.740,398.249,164.751,58.569,160.253
C02919=1014.687,-119.490,398.241,164.753,58.563,160.253
C02920=1014.693,-119.240,398.234,164.756,58.558,160.253
C02921=1014.697,-118.991,398.227,164.759,58.552,160.252
C02922=1014.701,-118.741,398.220,164.762,58.546,160.252
C02923=1014.707,-118.459,398.211,164.765,58.538,160.252
C02924=1014.712,-118.177,398.203,164.768,58.532,160.251
C02925=1014.717,-117.895,398.195,164.771,58.525,160.251
C02926=1014.723,-117.614,398.187,164.773,58.519,160.250
C02927=1014.728,-117.364,398.180,164.777,58.513,160.250
C02928=1014.733,-117.114,398.172,164.779,58.507,160.250
C02929=1014.737,-116.864,398.165,164.782,58.501,160.249
C02930=1014.742,-116.614,398.159,164.785,58.494,160.249
C02931=1014.747,-116.364,398.151,164.787,58.488,160.249
C02932=1014.751,-116.114,398.143,164.790,58.482,160.248
C02933=1014.755,-115.865,398.136,164.793,58.476,160.248
C02934=1014.761,-115.615,398.129,164.796,58.471,160.248
C02935=1014.765,-115.365,398.121,164.799,58.465,160.248
C02936=1014.770,-115.115,398.114,164.801,58.459,160.247
C02937=1014.775,-114.865,398.106,164.804,58.453,160.247
C02938=1014.779,-114.615,398.099,164.807,58.447,160.247
C02939=1014.785,-114.365,398.092,164.809,58.441,160.246
C02940=1014.789,-114.116,398.084,164.813,58.434,160.246
C02941=1014.794,-113.866,398.077,164.815,58.428,160.246
C02942=1014.799,-113.616,398.069,164.817,58.422,160.245
C02943=1014.803,-113.366,398.062,164.821,58.416,160.245
C02944=1014.808,-113.116,398.054,164.823,58.410,160.245
C02945=1014.812,-112.866,398.047,164.825,58.404,160.244
C02946=1014.817,-112.617,398.039,164.829,58.398,160.244
C02947=1014.822,-112.366,398.032,164.831,58.392,160.243
C02948=1014.827,-112.117,398.024,164.834,58.386,160.243
C02949=1014.832,-111.867,398.016,164.837,58.380,160.243
C02950=1014.836,-111.618,398.009,164.839,58.374,160.242
C02951=1014.841,-111.367,398.001,164.842,58.368,160.242
C02952=1014.846,-111.118,397.994,164.845,58.361,160.242
C02953=1014.850,-110.868,397.986,164.848,58.355,160.241
C02954=1014.855,-110.618,397.978,164.851,58.349,160.241
C02955=1014.860,-110.368,397.972,164.853,58.343,160.241
C02956=1014.865,-110.119,397.963,164.856,58.337,160.240
C02957=1014.870,-109.869,397.956,164.859,58.331,160.240
C02958=1014.875,-109.619,397.948,164.862,58.325,160.240
C02959=1014.879,-109.369,397.941,164.864,58.318,160.239
C02960=1014.884,-109.119,397.933,164.867,58.312,160.239
C02961=1014.888,-108.869,397.925,164.869,58.306,160.238
C02962=1014.893,-108.619,397.917,164.873,58.300,160.238
C02963=1014.898,-108.370,397.909,164.875,58.294,160.238
C02964=1014.904,-108.120,397.902,164.878,58.287,160.238
C02965=1014.908,-107.870,397.895,164.881,58.281,160.237
C02966=1014.913,-107.620,397.887,164.884,58.275,160.237
C02967=1014.918,-107.371,397.879,164.886,58.268,160.236
C02968=1014.922,-107.120,397.871,164.888,58.262,160.236
C02969=1014.927,-106.871,397.864,164.892,58.256,160.236
C02970=1014.932,-106.621,397.855,164.894,58.250,160.235
C02971=1014.936,-106.371,397.848,164.898,58.244,160.235
C02972=1014.941,-106.121,397.840,164.900,58.238,160.235
C02973=1014.946,-105.871,397.831,164.902,58.232,160.234
C02974=1014.950,-105.621,397.824,164.906,58.226,160.234
C02975=1014.955,-105.371,397.816,164.908,58.220,160.233
C02976=1014.960,-105.122,397.808,164.911,58.213,160.233
C02977=1014.965,-104.872,397.800,164.914,58.207,160.233
C02978=1014.970,-104.623,397.792,164.917,58.200,160.232
C02979=1014.974,-104.372,397.784,164.919,58.194,160.232
C02980=1014.979,-104.122,397.776,164.923,58.188,160.232
C02981=1014.984,-103.873,397.768,164.925,58.182,160.231
C02982=1014.989,-103.623,397.760,164.928,58.176,160.231
C02983=1014.994,-103.374,397.752,164.931,58.169,160.230
C02984=1014.999,-103.123,397.745,164.933,58.163,160.230
C02985=1015.004,-102.874,397.736,164.936,58.157,160.230
C02986=1015.008,-102.624,397.728,164.939,58.151,160.229
C02987=1015.013,-102.342,397.720,164.942,58.144,160.229
C02988=1015.019,-102.061,397.710,164.946,58.136,160.229
C02989=1015.024,-101.779,397.702,164.948,58.129,160.228
C02990=1015.029,-101.497,397.692,164.951,58.122,160.227
C02991=1015.034,-101.247,397.684,164.955,58.116,160.227
C02992=1015.040,-100.997,397.676,164.957,58.110,160.227
C02993=1015.044,-100.748,397.668,164.960,58.103,160.226
C02994=1015.049,-100.498,397.660,164.962,58.097,160.226
C02995=1015.054,-100.248,397.652,164.966,58.091,160.226
C02996=1015.059,-99.999,397.644,164.968,58.084,160.225
C02997=1015.064,-99.749,397.635,164.971,58.078,160.225
C02998=1015.068,-99.498,397.627,164.974,58.072,160.224
C02999=1015.074,-99.249,397.618,164.976,58.065,160.224
C03000=1015.078,-98.999,397.611,164.979,58.059,160.223
C03001=1015.083,-98.749,397.603,164.982,58.052,160.223
C03002=1015.088,-98.499,397.595,164.985,58.045,160.223
C03003=1015.093,-98.250,397.587,164.988,58.040,160.222
C03004=1015.098,-98.000,397.578,164.991,58.033,160.222
C03005=1015.102,-97.749,397.570,164.993,58.027,160.221
C03006=1015.108,-97.500,397.561,164.996,58.020,160.221
C03007=1015.112,-97.251,397.553,164.999,58.014,160.221
C03008=1015.117,-97.001,397.544,165.002,58.008,160.221
C03009=1015.122,-96.750,397.536,165.005,58.002,160.220
C03010=1015.127,-96.501,397.528,165.006,57.995,160.219
C03011=1015.132,-96.251,397.519,165.010,57.989,160.219
C03012=1015.136,-96.002,397.511,165.012,57.983,160.219
C03013=1015.140,-95.751,397.502,165.016,57.977,160.219
C03014=1015.146,-95.501,397.494,165.018,57.971,160.218
C03015=1015.151,-95.252,397.485,165.021,57.964,160.218
C03016=1015.155,-95.002,397.477,165.024,57.958,160.217
C03017=1015.160,-94.753,397.468,165.027,57.952,160.217
C03018=1015.165,-94.502,397.459,165.029,57.945,160.216
C03019=1015.170,-94.252,397.451,165.032,57.939,160.216
C03020=1015.175,-94.002,397.443,165.035,57.933,160.216
C03021=1015.179,-93.752,397.434,165.038,57.927,160.215
C03022=1015.184,-93.503,397.426,165.041,57.920,160.215
C03023=1015.189,-93.253,397.417,165.044,57.914,160.214
C03024=1015.194,-93.004,397.408,165.047,57.907,160.214
C03025=1015.199,-92.754,397.400,165.049,57.901,160.213
C03026=1015.204,-92.504,397.390,165.052,57.894,160.213
C03027=1015.209,-92.254,397.383,165.054,57.888,160.213
C03028=1015.213,-92.005,397.375,165.058,57.881,160.212
C03029=1015.218,-91.755,397.366,165.060,57.876,160.212
C03030=1015.223,-91.505,397.357,165.063,57.868,160.211
C03031=1015.228,-91.255,397.348,165.066,57.862,160.211
C03032=1015.233,-91.005,397.339,165.068,57.856,160.210
C03033=1015.238,-90.755,397.331,165.072,57.849,160.210
C03034=1015.243,-90.505,397.322,165.074,57.843,160.210
C03035=1015.248,-90.256,397.313,165.077,57.836,160.209
C03036=1015.253,-90.006,397.304,165.081,57.830,160.209
C03037=1015.257,-89.757,397.296,165.082,57.823,160.208
C03038=1015.262,-89.507,397.288,165.086,57.817,160.208
C03039=1015.267,-89.257,397.279,165.089,57.810,160.208
C03040=1015.272,-89.007,397.270,165.091,57.804,160.207
C03041=1015.277,-88.757,397.261,165.094,57.797,160.207
C03042=1015.282,-88.507,397.253,165.097,57.791,160.206
C03043=1015.287,-88.257,397.244,165.099,57.784,160.206
C03044=1015.292,-88.008,397.235,165.103,57.778,160.206
C03045=1015.297,-87.758,397.227,165.105,57.771,160.205
C03046=1015.302,-87.508,397.217,165.108,57.765,160.205
C03047=1015.307,-87.258,397.209,165.111,57.758,160.204
C03048=1015.311,-87.008,397.200,165.113,57.751,160.203
C03049=1015.317,-86.758,397.191,165.117,57.745,160.203
C03050=1015.322,-86.509,397.183,165.119,57.738,160.203
C03051=1015.328,-86.230,397.173,165.122,57.731,160.202
C03052=1015.333,-85.950,397.163,165.125,57.724,160.202
C03053=1015.339,-85.670,397.153,165.129,57.716,160.201
C03054=1015.345,-85.391,397.143,165.132,57.709,160.200
C03055=1015.349,-85.141,397.134,165.135,57.702,160.200
C03056=1015.354,-84.891,397.125,165.138,57.695,160.200
C03057=1015.359,-84.641,397.116,165.140,57.689,160.199
C03058=1015.364,-84.391,397.108,165.143,57.682,160.199
C03059=1015.369,-84.141,397.099,165.146,57.675,160.198
C03060=1015.374,-83.891,397.090,165.149,57.668,160.198
C03061=1015.379,-83.642,397.082,165.152,57.662,160.197
C03062=1015.384,-83.392,397.072,165.155,57.655,160.197
C03063=1015.390,-83.099,397.062,165.158,57.647,160.196
C03064=1015.396,-82.805,397.051,165.161,57.639,160.196
C03065=1015.402,-82.512,397.041,165.164,57.632,160.195
C03066=1015.408,-82.218,397.031,165.168,57.624,160.195
C03067=1015.413,-81.968,397.022,165.171,57.617,160.194
///RCONF 1,0,0,0,0,0,0,0,0,0,0,0,0,0,0,0,0,0,0,0,0,0,0,0
C03068=1015.418,-81.718,397.013,165.174,57.610,160.193
C03069=1015.423,-81.468,397.004,165.176,57.604,160.193
C03070=1015.428,-81.218,396.994,165.179,57.597,160.193
C03071=1015.433,-80.969,396.986,165.182,57.590,160.192
C03072=1015.439,-80.719,396.978,165.185,57.583,160.192
C03073=1015.443,-80.469,396.968,165.188,57.576,160.191
C03074=1015.448,-80.220,396.959,165.190,57.570,160.191
C03075=1015.453,-79.970,396.950,165.193,57.563,160.190
C03076=1015.458,-79.719,396.941,165.197,57.557,160.190
C03077=1015.463,-79.470,396.931,165.199,57.550,160.189
C03078=1015.468,-79.220,396.922,165.202,57.543,160.189
C03079=1015.473,-78.971,396.913,165.205,57.537,160.188
C03080=1015.478,-78.721,396.904,165.207,57.530,160.188
C03081=1015.483,-78.472,396.894,165.210,57.523,160.187
C03082=1015.488,-78.221,396.885,165.213,57.517,160.187
C03083=1015.493,-77.971,396.876,165.216,57.510,160.186
C03084=1015.498,-77.721,396.866,165.218,57.503,160.186
C03085=1015.503,-77.472,396.858,165.222,57.497,160.185
C03086=1015.508,-77.222,396.848,165.225,57.490,160.185
C03087=1015.512,-76.972,396.839,165.227,57.483,160.184
C03088=1015.519,-76.722,396.829,165.230,57.477,160.184
C03089=1015.523,-76.472,396.820,165.233,57.470,160.183
C03090=1015.528,-76.223,396.810,165.236,57.463,160.183
C03091=1015.533,-75.973,396.802,165.238,57.457,160.182
C03092=1015.538,-75.724,396.792,165.241,57.450,160.182
C03093=1015.543,-75.473,396.782,165.244,57.443,160.181
C03094=1015.548,-75.224,396.773,165.247,57.436,160.181
C03095=1015.553,-74.974,396.764,165.249,57.430,160.180
C03096=1015.558,-74.725,396.754,165.253,57.423,160.180
C03097=1015.564,-74.474,396.744,165.256,57.416,160.180
C03098=1015.568,-74.224,396.735,165.258,57.410,160.179
C03099=1015.573,-73.975,396.725,165.261,57.404,160.179
C03100=1015.578,-73.726,396.716,165.264,57.397,160.178
C03101=1015.583,-73.475,396.706,165.266,57.391,160.178
C03102=1015.588,-73.226,396.696,165.269,57.384,160.177
C03103=1015.593,-72.976,396.687,165.272,57.377,160.177
C03104=1015.598,-72.726,396.676,165.275,57.371,160.176
C03105=1015.603,-72.476,396.667,165.278,57.364,160.176
C03106=1015.607,-72.227,396.658,165.281,57.358,160.175
C03107=1015.612,-71.977,396.648,165.283,57.351,160.175
C03108=1015.618,-71.727,396.638,165.286,57.344,160.174
C03109=1015.622,-71.478,396.628,165.290,57.338,160.174
C03110=1015.627,-71.228,396.619,165.292,57.331,160.173
C03111=1015.633,-70.986,396.609,165.295,57.325,160.173
C03112=1015.637,-70.744,396.600,165.297,57.318,160.172
C03113=1015.642,-70.502,396.590,165.301,57.312,160.172
C03114=1015.646,-70.261,396.580,165.303,57.306,160.171
C03115=1015.651,-70.019,396.571,165.306,57.299,160.171
C03116=1015.656,-69.777,396.561,165.308,57.293,160.170
C03117=1015.661,-69.535,396.552,165.311,57.286,160.170
C03118=1015.666,-69.294,396.542,165.313,57.280,160.169
C03119=1015.671,-69.044,396.533,165.316,57.273,160.169
C03120=1015.676,-68.795,396.523,165.319,57.266,160.168
C03121=1015.681,-68.545,396.513,165.322,57.260,160.168
C03122=1015.686,-68.295,396.504,165.325,57.253,160.167
C03123=1015.690,-68.044,396.493,165.328,57.246,160.167
C03124=1015.695,-67.795,396.483,165.331,57.239,160.166
C03125=1015.700,-67.545,396.473,165.333,57.233,160.166
C03126=1015.706,-67.295,396.463,165.336,57.226,160.165
C03127=1015.710,-67.046,396.453,165.339,57.219,160.165
C03128=1015.715,-66.796,396.444,165.342,57.212,160.164
C03129=1015.721,-66.546,396.433,165.344,57.206,160.164
C03130=1015.726,-66.297,396.424,165.347,57.199,160.163
C03131=1015.731,-66.047,396.413,165.351,57.193,160.163
C03132=1015.736,-65.797,396.404,165.354,57.186,160.162
C03133=1015.741,-65.547,396.393,165.356,57.179,160.162
C03134=1015.746,-65.298,396.384,165.359,57.172,160.161
C03135=1015.751,-65.048,396.374,165.362,57.165,160.161
C03136=1015.756,-64.798,396.364,165.364,57.158,160.160
C03137=1015.761,-64.549,396.354,165.366,57.152,160.159
C03138=1015.767,-64.299,396.344,165.369,57.145,160.159
C03139=1015.771,-64.049,396.334,165.373,57.139,160.159
C03140=1015.777,-63.799,396.324,165.376,57.132,160.158
C03141=1015.782,-63.550,396.314,165.379,57.125,160.158
C03142=1015.787,-63.300,396.304,165.381,57.118,160.157
C03143=1015.792,-63.050,396.294,165.384,57.111,160.156
C03144=1015.797,-62.800,396.284,165.387,57.104,160.156
C03145=1015.802,-62.551,396.274,165.390,57.097,160.155
C03146=1015.808,-62.301,396.264,165.393,57.090,160.155
C03147=1015.812,-62.051,396.254,165.395,57.084,160.154
C03148=1015.818,-61.801,396.244,165.398,57.077,160.154
C03149=1015.823,-61.552,396.234,165.401,57.070,160.153
C03150=1015.828,-61.302,396.224,165.404,57.063,160.153
C03151=1015.833,-61.052,396.214,165.407,57.056,160.152
C03152=1015.838,-60.802,396.204,165.410,57.049,160.151
C03153=1015.843,-60.553,396.194,165.412,57.042,160.151
C03154=1015.848,-60.302,396.184,165.415,57.035,160.150
C03155=1015.853,-60.053,396.174,165.418,57.028,160.150
C03156=1015.859,-59.804,396.163,165.421,57.021,160.149
C03157=1015.864,-59.553,396.153,165.424,57.014,160.149
C03158=1015.869,-59.304,396.143,165.427,57.007,160.148
C03159=1015.874,-59.054,396.133,165.430,57.001,160.148
C03160=1015.879,-58.804,396.123,165.432,56.993,160.147
C03161=1015.885,-58.554,396.113,165.434,56.986,160.146
C03162=1015.889,-58.305,396.103,165.437,56.979,160.146
C03163=1015.895,-58.055,396.092,165.440,56.972,160.145
C03164=1015.901,-57.805,396.082,165.443,56.965,160.145
C03165=1015.905,-57.556,396.072,165.446,56.959,160.144
C03166=1015.911,-57.306,396.062,165.449,56.952,160.143
C03167=1015.916,-57.056,396.052,165.452,56.945,160.143
C03168=1015.921,-56.807,396.041,165.455,56.937,160.142
C03169=1015.927,-56.557,396.031,165.458,56.930,160.142
C03170=1015.932,-56.307,396.021,165.460,56.923,160.141
C03171=1015.937,-56.057,396.011,165.463,56.917,160.140
C03172=1015.942,-55.807,396.000,165.466,56.910,160.140
C03173=1015.947,-55.558,395.990,165.468,56.902,160.139
C03174=1015.952,-55.308,395.980,165.471,56.895,160.139
C03175=1015.958,-55.058,395.970,165.474,56.888,160.138
C03176=1015.963,-54.809,395.959,165.477,56.881,160.138
C03177=1015.968,-54.559,395.949,165.480,56.874,160.137
C03178=1015.974,-54.309,395.939,165.483,56.866,160.136
C03179=1015.979,-54.032,395.928,165.485,56.859,160.135
C03180=1015.986,-53.756,395.916,165.489,56.851,160.135
C03181=1015.991,-53.480,395.905,165.493,56.843,160.134
C03182=1015.997,-53.203,395.893,165.495,56.836,160.134
C03183=1016.002,-52.954,395.883,165.498,56.828,160.133
C03184=1016.008,-52.703,395.873,165.501,56.821,160.132
C03185=1016.013,-52.454,395.862,165.504,56.814,160.132
C03186=1016.019,-52.204,395.852,165.506,56.806,160.131
C03187=1016.024,-51.954,395.842,165.509,56.800,160.130
C03188=1016.029,-51.705,395.831,165.512,56.793,160.130
C03189=1016.035,-51.455,395.821,165.515,56.785,160.129
C03190=1016.039,-51.205,395.811,165.518,56.778,160.129
C03191=1016.045,-50.956,395.800,165.521,56.771,160.128
C03192=1016.050,-50.706,395.790,165.524,56.764,160.128
C03193=1016.055,-50.456,395.778,165.526,56.758,160.127
C03194=1016.060,-50.206,395.768,165.529,56.751,160.126
C03195=1016.065,-49.956,395.757,165.532,56.744,160.126
C03196=1016.071,-49.707,395.746,165.535,56.737,160.125
C03197=1016.075,-49.457,395.735,165.538,56.730,160.125
C03198=1016.081,-49.207,395.725,165.540,56.723,160.124
C03199=1016.086,-48.957,395.713,165.542,56.716,160.123
C03200=1016.091,-48.708,395.703,165.545,56.709,160.123
C03201=1016.096,-48.458,395.692,165.548,56.702,160.122
C03202=1016.101,-48.208,395.682,165.551,56.695,160.122
C03203=1016.106,-47.958,395.670,165.555,56.688,160.121
C03204=1016.112,-47.709,395.659,165.556,56.682,160.120
C03205=1016.116,-47.459,395.649,165.560,56.675,160.120
C03206=1016.122,-47.209,395.638,165.563,56.668,160.119
C03207=1016.127,-46.960,395.627,165.565,56.660,160.119
C03208=1016.132,-46.710,395.616,165.568,56.653,160.118
C03209=1016.137,-46.460,395.605,165.571,56.646,160.118
C03210=1016.142,-46.211,395.594,165.573,56.640,160.117
C03211=1016.147,-45.961,395.583,165.576,56.633,160.116
C03212=1016.153,-45.711,395.573,165.579,56.625,160.115
C03213=1016.158,-45.461,395.561,165.582,56.618,160.115
C03214=1016.164,-45.212,395.550,165.585,56.611,160.114
C03215=1016.169,-44.962,395.540,165.588,56.605,160.114
C03216=1016.174,-44.712,395.529,165.591,56.598,160.113
C03217=1016.179,-44.463,395.518,165.592,56.590,160.112
C03218=1016.184,-44.213,395.507,165.595,56.584,160.112
C03219=1016.190,-43.964,395.496,165.599,56.577,160.111
C03220=1016.195,-43.713,395.485,165.602,56.570,160.111
C03221=1016.200,-43.464,395.474,165.604,56.562,160.110
C03222=1016.205,-43.214,395.463,165.607,56.555,160.109
C03223=1016.211,-42.965,395.452,165.610,56.548,160.109
C03224=1016.216,-42.714,395.441,165.613,56.541,160.108
C03225=1016.221,-42.465,395.430,165.616,56.534,160.108
C03226=1016.226,-42.215,395.419,165.618,56.527,160.107
C03227=1016.232,-41.966,395.408,165.621,56.520,160.106
C03228=1016.237,-41.716,395.397,165.623,56.513,160.106
C03229=1016.242,-41.467,395.386,165.626,56.506,160.105
C03230=1016.247,-41.216,395.375,165.629,56.499,160.105
C03231=1016.253,-40.967,395.364,165.632,56.491,160.104
C03232=1016.258,-40.717,395.353,165.635,56.484,160.103
C03233=1016.264,-40.468,395.342,165.638,56.477,160.102
C03234=1016.269,-40.218,395.330,165.641,56.470,160.102
C03235=1016.274,-39.968,395.320,165.644,56.463,160.101
C03236=1016.279,-39.719,395.308,165.646,56.455,160.101
C03237=1016.285,-39.468,395.298,165.649,56.449,160.100
C03238=1016.290,-39.219,395.287,165.651,56.442,160.099
C03239=1016.295,-38.969,395.275,165.654,56.435,160.099
C03240=1016.300,-38.719,395.264,165.657,56.428,160.098
C03241=1016.306,-38.470,395.252,165.660,56.421,160.097
C03242=1016.311,-38.220,395.241,165.663,56.414,160.097
C03243=1016.316,-37.943,395.228,165.666,56.406,160.096
C03244=1016.322,-37.668,395.216,165.668,56.399,160.095
C03245=1016.327,-37.391,395.203,165.672,56.391,160.095
C03246=1016.334,-37.115,395.190,165.674,56.383,160.094
C03247=1016.339,-36.865,395.178,165.677,56.376,160.093
C03248=1016.344,-36.616,395.167,165.680,56.369,160.093
C03249=1016.350,-36.366,395.156,165.683,56.362,160.092
C03250=1016.355,-36.116,395.144,165.686,56.355,160.092
C03251=1016.360,-35.867,395.133,165.689,56.348,160.091
C03252=1016.365,-35.617,395.122,165.691,56.341,160.090
C03253=1016.370,-35.367,395.111,165.694,56.334,160.089
C03254=1016.375,-35.117,395.099,165.697,56.327,160.089
C03255=1016.380,-34.868,395.088,165.700,56.320,160.088
C03256=1016.386,-34.618,395.076,165.703,56.312,160.088
C03257=1016.391,-34.369,395.065,165.706,56.306,160.087
C03258=1016.396,-34.119,395.053,165.709,56.299,160.087
C03259=1016.401,-33.869,395.042,165.710,56.292,160.086
C03260=1016.406,-33.620,395.030,165.713,56.285,160.085
C03261=1016.412,-33.370,395.018,165.716,56.277,160.084
C03262=1016.417,-33.121,395.007,165.719,56.270,160.084
C03263=1016.423,-32.870,394.995,165.722,56.263,160.083
C03264=1016.428,-32.621,394.984,165.725,56.256,160.082
C03265=1016.433,-32.371,394.972,165.728,56.249,160.082
C03266=1016.438,-32.122,394.960,165.730,56.241,160.081
C03267=1016.444,-31.872,394.949,165.733,56.234,160.081
C03268=1016.449,-31.622,394.938,165.735,56.228,160.080
C03269=1016.454,-31.373,394.926,165.738,56.220,160.079
C03270=1016.459,-31.123,394.915,165.741,56.214,160.078
C03271=1016.465,-30.874,394.903,165.744,56.206,160.078
C03272=1016.471,-30.623,394.891,165.747,56.199,160.077
C03273=1016.476,-30.374,394.880,165.749,56.191,160.076
C03274=1016.481,-30.124,394.868,165.752,56.185,160.076
C03275=1016.486,-29.875,394.856,165.755,56.177,160.075
C03276=1016.492,-29.625,394.845,165.758,56.170,160.075
C03277=1016.497,-29.375,394.834,165.761,56.163,160.074
C03278=1016.503,-29.125,394.821,165.764,56.156,160.073
C03279=1016.508,-28.876,394.810,165.765,56.149,160.072
C03280=1016.513,-28.626,394.798,165.768,56.142,160.072
C03281=1016.519,-28.377,394.787,165.771,56.134,160.071
C03282=1016.524,-28.127,394.775,165.774,56.127,160.070
C03283=1016.529,-27.877,394.764,165.777,56.120,160.070
C03284=1016.535,-27.627,394.751,165.780,56.113,160.069
C03285=1016.540,-27.378,394.740,165.782,56.105,160.068
C03286=1016.545,-27.128,394.728,165.785,56.098,160.068
C03287=1016.551,-26.878,394.716,165.789,56.092,160.067
C03288=1016.556,-26.629,394.704,165.790,56.084,160.066
C03289=1016.561,-26.379,394.692,165.793,56.078,160.066
C03290=1016.566,-26.130,394.680,165.796,56.071,160.065
C03291=1016.571,-25.880,394.669,165.799,56.063,160.064
C03292=1016.577,-25.630,394.656,165.802,56.056,160.064
C03293=1016.581,-25.380,394.644,165.804,56.049,160.063
C03294=1016.587,-25.131,394.632,165.807,56.042,160.062
C03295=1016.592,-24.881,394.620,165.809,56.035,160.061
C03296=1016.598,-24.631,394.608,165.812,56.028,160.061
C03297=1016.603,-24.381,394.596,165.816,56.021,160.060
C03298=1016.608,-24.132,394.584,165.818,56.014,160.060
C03299=1016.613,-23.883,394.572,165.820,56.007,160.059
C03300=1016.619,-23.632,394.560,165.823,56.000,160.058
C03301=1016.624,-23.383,394.548,165.826,55.993,160.058
C03302=1016.629,-23.133,394.536,165.829,55.985,160.057
C03303=1016.634,-22.884,394.524,165.832,55.978,160.056
C03304=1016.640,-22.634,394.512,165.834,55.971,160.055
C03305=1016.645,-22.385,394.500,165.837,55.964,160.055
C03306=1016.650,-22.135,394.487,165.839,55.957,160.054
C03307=1016.656,-21.858,394.474,165.843,55.949,160.053
C03308=1016.662,-21.580,394.461,165.846,55.941,160.053
C03309=1016.668,-21.303,394.447,165.849,55.933,160.052
C03310=1016.675,-21.026,394.434,165.852,55.925,160.051
C03311=1016.680,-20.776,394.422,165.854,55.918,160.050
C03312=1016.685,-20.527,394.410,165.857,55.911,160.050
C03313=1016.691,-20.277,394.397,165.860,55.904,160.049
C03314=1016.695,-20.027,394.385,165.863,55.896,160.048
C03315=1016.700,-19.778,394.373,165.866,55.890,160.048
C03316=1016.706,-19.528,394.361,165.868,55.882,160.047
C03317=1016.711,-19.278,394.349,165.871,55.874,160.046
C03318=1016.717,-19.029,394.337,165.874,55.868,160.046
C03319=1016.722,-18.779,394.324,165.877,55.860,160.045
C03320=1016.728,-18.530,394.312,165.879,55.854,160.044
C03321=1016.733,-18.280,394.301,165.881,55.846,160.043
C03322=1016.739,-18.030,394.288,165.884,55.839,160.042
C03323=1016.744,-17.781,394.276,165.887,55.832,160.042
C03324=1016.750,-17.530,394.264,165.890,55.824,160.041
C03325=1016.754,-17.281,394.251,165.892,55.817,160.040
C03326=1016.759,-17.032,394.239,165.896,55.810,160.040
C03327=1016.765,-16.782,394.227,165.898,55.802,160.039
C03328=1016.770,-16.532,394.215,165.901,55.795,160.038
C03329=1016.776,-16.282,394.203,165.904,55.788,160.038
C03330=1016.782,-16.033,394.190,165.907,55.780,160.037
C03331=1016.787,-15.784,394.178,165.909,55.774,160.036
C03332=1016.792,-15.534,394.165,165.911,55.767,160.035
C03333=1016.797,-15.284,394.153,165.915,55.760,160.035
C03334=1016.803,-15.035,394.140,165.917,55.752,160.034
C03335=1016.808,-14.785,394.128,165.920,55.745,160.033
C03336=1016.814,-14.535,394.115,165.922,55.738,160.033
C03337=1016.818,-14.286,394.102,165.925,55.731,160.032
C03338=1016.824,-14.036,394.090,165.928,55.724,160.031
C03339=1016.830,-13.787,394.078,165.931,55.717,160.031
C03340=1016.834,-13.537,394.065,165.934,55.710,160.030
C03341=1016.840,-13.287,394.052,165.936,55.702,160.029
C03342=1016.845,-13.038,394.040,165.938,55.696,160.028
C03343=1016.851,-12.788,394.027,165.941,55.688,160.028
C03344=1016.856,-12.539,394.015,165.944,55.681,160.027
C03345=1016.861,-12.288,394.001,165.947,55.674,160.026
C03346=1016.866,-12.039,393.989,165.950,55.667,160.026
C03347=1016.872,-11.789,393.977,165.953,55.660,160.025
C03348=1016.877,-11.540,393.964,165.954,55.652,160.024
C03349=1016.883,-11.290,393.951,165.957,55.646,160.023
C03350=1016.888,-11.041,393.939,165.960,55.638,160.023
C03351=1016.893,-10.791,393.926,165.963,55.631,160.022
C03352=1016.898,-10.541,393.914,165.966,55.624,160.021
C03353=1016.904,-10.291,393.901,165.968,55.616,160.020
C03354=1016.909,-10.042,393.889,165.972,55.610,160.020
C03355=1016.915,-9.792,393.876,165.973,55.602,160.019
C03356=1016.919,-9.543,393.863,165.976,55.595,160.018
C03357=1016.925,-9.293,393.851,165.979,55.588,160.018
C03358=1016.931,-9.044,393.838,165.982,55.581,160.017
C03359=1016.936,-8.793,393.825,165.984,55.573,160.016
C03360=1016.941,-8.544,393.813,165.988,55.566,160.016
C03361=1016.947,-8.295,393.799,165.990,55.559,160.015
C03362=1016.953,-8.045,393.787,165.992,55.552,160.014
C03363=1016.958,-7.796,393.775,165.995,55.544,160.013
C03364=1016.963,-7.545,393.761,165.998,55.538,160.012
C03365=1016.968,-7.296,393.749,166.000,55.530,160.012
C03366=1016.973,-7.046,393.736,166.003,55.523,160.011
C03367=1016.979,-6.797,393.724,166.006,55.515,160.010
C03368=1016.985,-6.548,393.711,166.009,55.508,160.010
C03369=1016.990,-6.297,393.697,166.012,55.501,160.009
C03370=1016.995,-6.048,393.685,166.014,55.493,160.008
C03371=1017.002,-5.769,393.671,166.017,55.486,160.007
C03372=1017.008,-5.490,393.657,166.020,55.477,160.006
C03373=1017.014,-5.211,393.642,166.022,55.469,160.005
C03374=1017.019,-4.932,393.628,166.026,55.461,160.005
C03375=1017.025,-4.682,393.615,166.029,55.454,160.004
C03376=1017.031,-4.432,393.603,166.032,55.446,160.003
C03377=1017.036,-4.183,393.589,166.035,55.439,160.002
C03378=1017.041,-3.933,393.576,166.036,55.432,160.001
C03379=1017.046,-3.683,393.563,166.040,55.425,160.001
C03380=1017.052,-3.434,393.550,166.042,55.418,160.000
C03381=1017.057,-3.184,393.537,166.045,55.410,159.999
C03382=1017.062,-2.935,393.523,166.047,55.404,159.999
C03383=1017.067,-2.685,393.510,166.050,55.397,159.998
C03384=1017.073,-2.435,393.498,166.053,55.390,159.997
C03385=1017.078,-2.186,393.484,166.056,55.382,159.997
C03386=1017.083,-1.936,393.471,166.058,55.376,159.996
C03387=1017.089,-1.686,393.457,166.061,55.369,159.995
C03388=1017.094,-1.437,393.445,166.063,55.361,159.994
C03389=1017.099,-1.188,393.431,166.066,55.354,159.994
C03390=1017.105,-0.938,393.418,166.068,55.347,159.993
C03391=1017.110,-0.689,393.404,166.071,55.340,159.992
C03392=1017.115,-0.439,393.392,166.074,55.333,159.991
C03393=1017.121,-0.189,393.378,166.077,55.326,159.991
C03394=1017.126,0.061,393.365,166.080,55.319,159.990
C03395=1017.131,0.310,393.351,166.082,55.312,159.989
C03396=1017.136,0.560,393.338,166.084,55.304,159.988
C03397=1017.142,0.809,393.325,166.088,55.298,159.988
C03398=1017.147,1.059,393.312,166.090,55.290,159.987
C03399=1017.152,1.308,393.298,166.092,55.283,159.986
C03400=1017.158,1.559,393.285,166.095,55.276,159.985
C03401=1017.163,1.807,393.272,166.098,55.269,159.985
C03402=1017.168,2.057,393.259,166.101,55.261,159.984
C03403=1017.174,2.307,393.245,166.103,55.254,159.983
C03404=1017.179,2.556,393.231,166.105,55.248,159.982
C03405=1017.185,2.806,393.219,166.108,55.240,159.982
C03406=1017.190,3.055,393.205,166.111,55.233,159.981
C03407=1017.195,3.305,393.192,166.114,55.225,159.980
C03408=1017.201,3.555,393.178,166.117,55.218,159.980
C03409=1017.206,3.804,393.165,166.118,55.211,159.979
C03410=1017.211,4.054,393.152,166.121,55.204,159.978
C03411=1017.217,4.303,393.138,166.124,55.196,159.977
C03412=1017.222,4.554,393.125,166.127,55.190,159.976
C03413=1017.228,4.803,393.111,166.130,55.182,159.976
C03414=1017.233,5.052,393.098,166.133,55.175,159.975
C03415=1017.238,5.302,393.085,166.134,55.168,159.974
C03416=1017.244,5.551,393.071,166.137,55.160,159.973
C03417=1017.249,5.801,393.058,166.140,55.153,159.972
C03418=1017.255,6.050,393.045,166.143,55.146,159.972
C03419=1017.260,6.300,393.032,166.146,55.139,159.971
C03420=1017.265,6.550,393.018,166.148,55.131,159.970
C03421=1017.271,6.800,393.004,166.150,55.124,159.969
C03422=1017.276,7.049,392.991,166.153,55.117,159.968
C03423=1017.282,7.298,392.977,166.156,55.109,159.968
C03424=1017.287,7.548,392.965,166.159,55.103,159.967
C03425=1017.292,7.797,392.951,166.162,55.095,159.966
C03426=1017.298,8.047,392.937,166.164,55.088,159.966
C03427=1017.303,8.297,392.924,166.167,55.080,159.965
C03428=1017.309,8.546,392.910,166.169,55.073,159.964
C03429=1017.315,8.796,392.897,166.172,55.066,159.963
C03430=1017.319,9.046,392.884,166.174,55.058,159.962
C03431=1017.325,9.295,392.870,166.177,55.051,159.961
C03432=1017.331,9.544,392.857,166.180,55.043,159.961
C03433=1017.337,9.794,392.843,166.183,55.036,159.960
C03434=1017.342,10.044,392.830,166.186,55.029,159.959
C03435=1017.348,10.325,392.814,166.188,55.021,159.958
C03436=1017.355,10.606,392.799,166.191,55.013,159.957
C03437=1017.360,10.887,392.783,166.194,55.004,159.956
C03438=1017.366,11.168,392.769,166.197,54.996,159.955
C03439=1017.372,11.418,392.755,166.200,54.988,159.955
C03440=1017.377,11.667,392.741,166.202,54.981,159.954
C03441=1017.383,11.916,392.728,166.205,54.974,159.953
C03442=1017.389,12.167,392.714,166.208,54.966,159.952
C03443=1017.394,12.416,392.701,166.210,54.959,159.951
C03444=1017.400,12.666,392.687,166.212,54.952,159.951
C03445=1017.406,12.915,392.673,166.215,54.944,159.950
C03446=1017.411,13.165,392.660,166.218,54.937,159.949
C03447=1017.417,13.414,392.646,166.221,54.929,159.948
C03448=1017.422,13.664,392.632,166.224,54.923,159.948
C03449=1017.427,13.914,392.618,166.226,54.916,159.947
C03450=1017.432,14.164,392.604,166.228,54.908,159.946
C03451=1017.437,14.413,392.591,166.231,54.901,159.945
C03452=1017.442,14.662,392.577,166.234,54.894,159.944
C03453=1017.448,14.912,392.563,166.237,54.886,159.944
C03454=1017.453,15.161,392.549,166.239,54.880,159.943
C03455=1017.459,15.411,392.535,166.242,54.872,159.942
C03456=1017.464,15.661,392.521,166.245,54.865,159.941
C03457=1017.470,15.910,392.508,166.247,54.858,159.940
C03458=1017.476,16.159,392.493,166.250,54.850,159.940
C03459=1017.481,16.409,392.479,166.252,54.843,159.939
C03460=1017.487,16.658,392.465,166.255,54.836,159.938
C03461=1017.491,16.908,392.451,166.257,54.828,159.937
C03462=1017.497,17.158,392.437,166.261,54.822,159.937
C03463=1017.502,17.407,392.423,166.263,54.814,159.936
C03464=1017.508,17.657,392.409,166.265,54.807,159.935
C03465=1017.513,17.906,392.395,166.268,54.800,159.934
C03466=1017.519,18.156,392.381,166.271,54.792,159.933
C03467=1017.524,18.406,392.368,166.274,54.785,159.933
C03468=1017.530,18.655,392.354,166.276,54.778,159.932
C03469=1017.535,18.905,392.340,166.278,54.771,159.931
C03470=1017.541,19.154,392.326,166.281,54.763,159.930
C03471=1017.546,19.404,392.311,166.284,54.756,159.929
C03472=1017.551,19.653,392.297,166.287,54.748,159.928
C03473=1017.557,19.903,392.283,166.289,54.742,159.928
C03474=1017.562,20.152,392.269,166.292,54.735,159.927
C03475=1017.567,20.402,392.255,166.294,54.727,159.926
C03476=1017.573,20.651,392.240,166.297,54.720,159.925
C03477=1017.578,20.901,392.226,166.299,54.713,159.924
C03478=1017.584,21.150,392.213,166.302,54.706,159.924
C03479=1017.588,21.400,392.198,166.305,54.698,159.923
C03480=1017.594,21.649,392.183,166.307,54.691,159.922
C03481=1017.600,21.899,392.170,166.310,54.683,159.921
C03482=1017.606,22.149,392.155,166.312,54.676,159.920
C03483=1017.611,22.399,392.142,166.315,54.669,159.920
C03484=1017.616,22.648,392.126,166.318,54.662,159.919
C03485=1017.622,22.897,392.112,166.321,54.655,159.918
C03486=1017.627,23.147,392.099,166.323,54.648,159.917
C03487=1017.633,23.397,392.085,166.325,54.641,159.916
C03488=1017.638,23.646,392.070,166.328,54.633,159.916
C03489=1017.643,23.895,392.056,166.331,54.626,159.915
C03490=1017.649,24.145,392.042,166.334,54.618,159.914
C03491=1017.654,24.394,392.027,166.336,54.611,159.913
C03492=1017.659,24.644,392.013,166.338,54.604,159.912
C03493=1017.665,24.893,391.999,166.341,54.597,159.912
C03494=1017.671,25.143,391.984,166.344,54.589,159.911
C03495=1017.676,25.393,391.970,166.347,54.582,159.910
C03496=1017.681,25.643,391.956,166.349,54.575,159.909
C03497=1017.687,25.891,391.941,166.351,54.568,159.908
C03498=1017.692,26.141,391.927,166.354,54.560,159.907
C03499=1017.698,26.424,391.911,166.358,54.552,159.907
C03500=1017.705,26.706,391.894,166.360,54.544,159.906
C03501=1017.711,26.988,391.878,166.363,54.535,159.905
C03502=1017.717,27.271,391.862,166.366,54.527,159.904
C03503=1017.722,27.520,391.847,166.369,54.520,159.903
C03504=1017.727,27.770,391.833,166.371,54.512,159.902
C03505=1017.733,28.020,391.818,166.373,54.505,159.901
C03506=1017.738,28.270,391.803,166.376,54.498,159.900
C03507=1017.744,28.519,391.789,166.379,54.491,159.900
C03508=1017.749,28.768,391.775,166.382,54.484,159.899
C03509=1017.755,29.018,391.760,166.384,54.477,159.898
C03510=1017.760,29.267,391.746,166.387,54.470,159.897
C03511=1017.766,29.517,391.730,166.390,54.462,159.897
C03512=1017.771,29.767,391.716,166.393,54.455,159.896
C03513=1017.776,30.016,391.701,166.394,54.448,159.895
C03514=1017.782,30.266,391.687,166.397,54.441,159.894
C03515=1017.787,30.515,391.672,166.400,54.433,159.893
C03516=1017.793,30.765,391.658,166.403,54.426,159.892
C03517=1017.798,31.014,391.643,166.405,54.419,159.891
C03518=1017.804,31.263,391.628,166.408,54.412,159.891
C03519=1017.808,31.513,391.614,166.410,54.404,159.890
C03520=1017.814,31.762,391.599,166.413,54.397,159.889
C03521=1017.819,32.013,391.584,166.415,54.390,159.888
C03522=1017.825,32.262,391.570,166.418,54.383,159.887
C03523=1017.830,32.511,391.555,166.421,54.375,159.887
C03524=1017.836,32.761,391.541,166.424,54.368,159.886
C03525=1017.841,33.010,391.526,166.425,54.361,159.885
C03526=1017.847,33.259,391.511,166.428,54.354,159.884
C03527=1017.852,33.509,391.496,166.431,54.346,159.883
C03528=1017.858,33.758,391.482,166.434,54.339,159.883
C03529=1017.862,34.008,391.467,166.436,54.332,159.882
C03530=1017.869,34.258,391.452,166.439,54.325,159.881
C03531=1017.874,34.507,391.437,166.442,54.317,159.880
C03532=1017.879,34.757,391.423,166.444,54.310,159.879
C03533=1017.884,35.006,391.408,166.447,54.303,159.878
C03534=1017.891,35.256,391.393,166.449,54.295,159.877
C03535=1017.896,35.505,391.378,166.451,54.288,159.876
C03536=1017.901,35.754,391.364,166.454,54.280,159.876
C03537=1017.907,36.004,391.348,166.457,54.273,159.875
C03538=1017.912,36.254,391.333,166.459,54.266,159.874
C03539=1017.917,36.503,391.319,166.462,54.259,159.873
C03540=1017.922,36.753,391.304,166.465,54.251,159.872
C03541=1017.928,37.003,391.289,166.468,54.244,159.872
C03542=1017.934,37.251,391.274,166.469,54.237,159.871
C03543=1017.939,37.501,391.259,166.472,54.230,159.870
C03544=1017.944,37.751,391.244,166.475,54.223,159.869
C03545=1017.949,38.001,391.229,166.477,54.216,159.868
C03546=1017.955,38.250,391.214,166.480,54.208,159.867
C03547=1017.961,38.500,391.199,166.483,54.201,159.867
C03548=1017.966,38.749,391.184,166.486,54.194,159.866
C03549=1017.971,38.998,391.168,166.488,54.187,159.865
C03550=1017.977,39.248,391.154,166.490,54.179,159.864
C03551=1017.982,39.497,391.138,166.493,54.172,159.863
C03552=1017.987,39.747,391.124,166.495,54.165,159.862
C03553=1017.993,39.997,391.108,166.498,54.158,159.862
C03554=1017.998,40.246,391.094,166.501,54.151,159.861
C03555=1018.003,40.495,391.079,166.504,54.143,159.860
C03556=1018.009,40.745,391.063,166.506,54.136,159.859
C03557=1018.014,40.994,391.048,166.509,54.129,159.858
C03558=1018.020,41.243,391.033,166.512,54.122,159.858
C03559=1018.026,41.493,391.018,166.514,54.114,159.857
C03560=1018.031,41.742,391.003,166.516,54.107,159.856
C03561=1018.036,41.992,390.987,166.519,54.100,159.855
C03562=1018.042,42.241,390.972,166.522,54.093,159.854
C03563=1018.047,42.524,390.955,166.524,54.085,159.853
C03564=1018.053,42.807,390.937,166.527,54.077,159.852
C03565=1018.059,43.089,390.920,166.530,54.068,159.851
C03566=1018.066,43.372,390.903,166.533,54.061,159.851
C03567=1018.071,43.621,390.887,166.536,54.054,159.850
C03568=1018.076,43.871,390.872,166.538,54.047,159.849
C03569=1018.081,44.120,390.857,166.541,54.040,159.848
C03570=1018.087,44.370,390.841,166.544,54.032,159.847
C03571=1018.092,44.619,390.826,166.546,54.025,159.846
C03572=1018.097,44.868,390.810,166.549,54.018,159.846
C03573=1018.102,45.118,390.794,166.552,54.011,159.845
C03574=1018.107,45.367,390.779,166.553,54.004,159.844
C03575=1018.113,45.617,390.763,166.556,53.997,159.843
C03576=1018.118,45.867,390.748,166.559,53.989,159.842
C03577=1018.123,46.116,390.733,166.561,53.982,159.841
C03578=1018.129,46.365,390.717,166.564,53.975,159.841
C03579=1018.134,46.615,390.702,166.567,53.968,159.840
C03580=1018.140,46.865,390.686,166.569,53.961,159.839
C03581=1018.145,47.114,390.671,166.572,53.954,159.838
C03582=1018.150,47.364,390.655,166.575,53.946,159.837
C03583=1018.156,47.612,390.639,166.577,53.939,159.836
C03584=1018.161,47.862,390.624,166.580,53.932,159.836
C03585=1018.166,48.112,390.609,166.582,53.925,159.835
C03586=1018.171,48.361,390.594,166.584,53.918,159.834
C03587=1018.177,48.610,390.577,166.587,53.911,159.833
C03588=1018.182,48.860,390.562,166.590,53.903,159.832
C03589=1018.188,49.110,390.547,166.592,53.896,159.831
C03590=1018.193,49.359,390.531,166.595,53.889,159.831
C03591=1018.199,49.608,390.515,166.598,53.882,159.830
C03592=1018.203,49.858,390.499,166.600,53.875,159.829
C03593=1018.209,50.108,390.484,166.603,53.868,159.828
C03594=1018.214,50.357,390.469,166.606,53.860,159.827
C03595=1018.220,50.606,390.452,166.609,53.853,159.827
C03596=1018.225,50.856,390.437,166.611,53.846,159.826
C03597=1018.231,51.106,390.422,166.613,53.839,159.825
C03598=1018.236,51.354,390.406,166.616,53.832,159.824
C03599=1018.242,51.604,390.390,166.618,53.825,159.823
C03600=1018.247,51.853,390.375,166.621,53.817,159.822
C03601=1018.253,52.103,390.359,166.624,53.810,159.821
C03602=1018.258,52.352,390.344,166.626,53.803,159.820
C03603=1018.263,52.602,390.328,166.629,53.795,159.820
C03604=1018.268,52.851,390.313,166.632,53.788,159.819
C03605=1018.274,53.101,390.297,166.634,53.781,159.818
C03606=1018.279,53.350,390.281,166.636,53.774,159.817
C03607=1018.285,53.600,390.265,166.639,53.767,159.816
C03608=1018.290,53.849,390.249,166.642,53.759,159.815
C03609=1018.295,54.099,390.234,166.645,53.752,159.815
C03610=1018.301,54.347,390.218,166.647,53.745,159.814
C03611=1018.306,54.597,390.202,166.650,53.737,159.813
C03612=1018.312,54.847,390.187,166.653,53.730,159.812
C03613=1018.317,55.096,390.171,166.655,53.723,159.811
C03614=1018.323,55.346,390.155,166.657,53.715,159.810
C03615=1018.328,55.595,390.140,166.660,53.708,159.809
C03616=1018.334,55.845,390.124,166.663,53.701,159.809
C03617=1018.339,56.094,390.109,166.665,53.694,159.808
C03618=1018.345,56.343,390.093,166.668,53.687,159.807
C03619=1018.351,56.593,390.077,166.670,53.679,159.806
C03620=1018.356,56.842,390.061,166.673,53.671,159.805
C03621=1018.361,57.092,390.045,166.675,53.665,159.804
C03622=1018.366,57.341,390.029,166.678,53.657,159.803
C03623=1018.372,57.591,390.014,166.681,53.650,159.803
C03624=1018.377,57.841,389.998,166.684,53.642,159.802
C03625=1018.383,58.089,389.982,166.687,53.635,159.801
C03626=1018.388,58.339,389.967,166.689,53.628,159.800
C03627=1018.395,58.621,389.949,166.692,53.620,159.799
C03628=1018.401,58.904,389.931,166.694,53.611,159.798
C03629=1018.407,59.186,389.912,166.698,53.603,159.797
C03630=1018.413,59.469,389.895,166.700,53.595,159.796
C03631=1018.419,59.718,389.879,166.703,53.587,159.795
C03632=1018.425,59.968,389.863,166.706,53.580,159.794
C03633=1018.430,60.217,389.847,166.709,53.572,159.793
C03634=1018.436,60.467,389.832,166.712,53.565,159.792
